   1:  PR[91,2] = PR[90,2] + -0.747;
   1:  PR[91,3] = PR[90,3] + 87.378;
   1:L PR[91] R[100]mm/sec CNT100;
   1:  PR[91,1] = PR[90,1] + -60.955;
   1:  PR[91,2] = PR[90,2] + -4.707;
   1:  PR[91,3] = PR[90,3] + 87.394;
   1:L PR[91] R[100]mm/sec CNT100;
   1:  PR[91,1] = PR[90,1] + -60.838;
   1:  PR[91,2] = PR[90,2] + -5.325;
   1:  PR[91,3] = PR[90,3] + 87.411;
   1:L PR[91] R[100]mm/sec CNT100;
   1:  PR[91,1] = PR[90,1] + -58.970;
   1:  PR[91,2] = PR[90,2] + -9.317;
   1:  PR[91,3] = PR[90,3] + 87.413;
   1:L PR[91] R[100]mm/sec CNT100;
   1:  PR[91,1] = PR[90,1] + -58.652;
   1:  PR[91,2] = PR[90,2] + -9.976;
   1:  PR[91,3] = PR[90,3] + 87.432;
   1:L PR[91] R[100]mm/sec CNT100;
   1:  PR[91,1] = PR[90,1] + -56.254;
   1:  PR[91,2] = PR[90,2] + -12.901;
   1:  PR[91,3] = PR[90,3] + 87.435;
   1:L PR[91] R[100]mm/sec CNT100;
   1:  PR[91,1] = PR[90,1] + -54.881;
   1:  PR[91,2] = PR[90,2] + -14.517;
   1:  PR[91,3] = PR[90,3] + 87.451;
   1:L PR[91] R[100]mm/sec CNT100;
   1:  PR[91,1] = PR[90,1] + -52.801;
   1:  PR[91,2] = PR[90,2] + -16.191;
   1:  PR[91,3] = PR[90,3] + 87.460;
   1:L PR[91] R[100]mm/sec CNT100;
   1:  PR[91,1] = PR[90,1] + -49.375;
   1:  PR[91,2] = PR[90,2] + -18.826;
   1:  PR[91,3] = PR[90,3] + 87.472;
   1:L PR[91] R[100]mm/sec CNT100;
   1:  PR[91,1] = PR[90,1] + -48.727;
   1:  PR[91,2] = PR[90,2] + -19.184;
   1:  PR[91,3] = PR[90,3] + 87.490;
   1:L PR[91] R[100]mm/sec CNT100;
   1:  PR[91,1] = PR[90,1] + -47.166;
   1:  PR[91,2] = PR[90,2] + -19.996;
   1:  PR[91,3] = PR[90,3] + 87.493;
   1:L PR[91] R[100]mm/sec CNT100;
   1:  PR[91,1] = PR[90,1] + -42.988;
   1:  PR[91,2] = PR[90,2] + -21.916;
   1:  PR[91,3] = PR[90,3] + 87.501;
   1:L PR[91] R[100]mm/sec CNT100;
   1:  PR[91,1] = PR[90,1] + -40.604;
   1:  PR[91,2] = PR[90,2] + -22.839;
   1:  PR[91,3] = PR[90,3] + 87.521;
   1:L PR[91] R[100]mm/sec CNT100;
   1:  PR[91,1] = PR[90,1] + -37.595;
   1:  PR[91,2] = PR[90,2] + -23.754;
   1:  PR[91,3] = PR[90,3] + 87.531;
   1:L PR[91] R[100]mm/sec CNT100;
   1:  PR[91,1] = PR[90,1] + -34.373;
   1:  PR[91,2] = PR[90,2] + -24.687;
   1:  PR[91,3] = PR[90,3] + 87.545;
   1:L PR[91] R[100]mm/sec CNT100;
   1:  PR[91,1] = PR[90,1] + -31.993;
   1:  PR[91,2] = PR[90,2] + -25.305;
   1:  PR[91,3] = PR[90,3] + 87.559;
   1:L PR[91] R[100]mm/sec CNT100;
   1:  PR[91,1] = PR[90,1] + -22.909;
   1:  PR[91,2] = PR[90,2] + -26.927;
   1:  PR[91,3] = PR[90,3] + 87.570;
   1:L PR[91] R[100]mm/sec CNT100;
   1:  PR[91,1] = PR[90,1] + -19.445;
   1:  PR[91,2] = PR[90,2] + -27.305;
   1:  PR[91,3] = PR[90,3] + 87.609;
   1:L PR[91] R[100]mm/sec CNT100;
   1:  PR[91,1] = PR[90,1] + -13.177;
   1:  PR[91,2] = PR[90,2] + -27.959;
   1:  PR[91,3] = PR[90,3] + 87.624;
   1:L PR[91] R[100]mm/sec CNT100;
   1:  PR[91,1] = PR[90,1] + -6.530;
   1:  PR[91,2] = PR[90,2] + -28.215;
   1:  PR[91,3] = PR[90,3] + 87.651;
   1:L PR[91] R[100]mm/sec CNT100;
   1:  PR[91,1] = PR[90,1] + -2.969;
   1:  PR[91,2] = PR[90,2] + -28.333;
   1:  PR[91,3] = PR[90,3] + 87.679;
   1:L PR[91] R[100]mm/sec CNT100;
   1:  PR[91,1] = PR[90,1] + 7.766;
   1:  PR[91,2] = PR[90,2] + -27.986;
   1:  PR[91,3] = PR[90,3] + 87.694;
   1:L PR[91] R[100]mm/sec CNT100;
   1:  PR[91,1] = PR[90,1] + 9.166;
   1:  PR[91,2] = PR[90,2] + -28.006;
   1:  PR[91,3] = PR[90,3] + 87.740;
   1:L PR[91] R[100]mm/sec CNT100;
   1:  PR[91,1] = PR[90,1] + 10.864;
   1:  PR[91,2] = PR[90,2] + -27.971;
   1:  PR[91,3] = PR[90,3] + 87.746;
   1:L PR[91] R[100]mm/sec CNT100;
   1:  PR[91,1] = PR[90,1] + 12.500;
   1:  PR[91,2] = PR[90,2] + -27.879;
   1:  PR[91,3] = PR[90,3] + 87.753;
   1:L PR[91] R[100]mm/sec CNT100;
   1:  PR[91,1] = PR[90,1] + 13.907;
   1:  PR[91,2] = PR[90,2] + -27.767;
   1:  PR[91,3] = PR[90,3] + 87.760;
   1:L PR[91] R[100]mm/sec CNT100;
   1:  PR[91,1] = PR[90,1] + 17.964;
   1:  PR[91,2] = PR[90,2] + -28.256;
   1:  PR[91,3] = PR[90,3] + 87.766;
   1:L PR[91] R[100]mm/sec CNT100;
   1:  PR[91,1] = PR[90,1] + 18.028;
   1:  PR[91,2] = PR[90,2] + -28.259;
   1:  PR[91,3] = PR[90,3] + 87.784;
   1:L PR[91] R[100]mm/sec CNT100;
   1:  PR[91,1] = PR[90,1] + 23.535;
   1:  PR[91,2] = PR[90,2] + -28.156;
   1:L PR[91] R[100]mm/sec CNT100;
   1:  PR[91,1] = PR[90,1] + 23.597;
   1:  PR[91,2] = PR[90,2] + -28.531;
   1:  PR[91,3] = PR[90,3] + 87.808;
   1:L PR[91] R[100]mm/sec CNT100;
   1:  PR[91,1] = PR[90,1] + 23.842;
   1:  PR[91,2] = PR[90,2] + -28.584;
   1:  PR[91,3] = PR[90,3] + 87.809;
   1:L PR[91] R[100]mm/sec CNT100;
   1:  PR[91,1] = PR[90,1] + 27.676;
   1:  PR[91,2] = PR[90,2] + -29.474;
   1:  PR[91,3] = PR[90,3] + 87.810;
   1:L PR[91] R[100]mm/sec CNT100;
   1:  PR[91,1] = PR[90,1] + 32.886;
   1:  PR[91,2] = PR[90,2] + -29.769;
   1:  PR[91,3] = PR[90,3] + 87.827;
   1:L PR[91] R[100]mm/sec CNT100;
   1:  PR[91,1] = PR[90,1] + 38.004;
   1:  PR[91,2] = PR[90,2] + -29.151;
   1:  PR[91,3] = PR[90,3] + 87.849;
   1:L PR[91] R[100]mm/sec CNT100;
   1:  PR[91,1] = PR[90,1] + 42.904;
   1:  PR[91,2] = PR[90,2] + -27.658;
   1:  PR[91,3] = PR[90,3] + 87.871;
   1:L PR[91] R[100]mm/sec CNT100;
   1:  PR[91,1] = PR[90,1] + 47.549;
   1:  PR[91,2] = PR[90,2] + -25.414;
   1:  PR[91,3] = PR[90,3] + 87.893;
   1:L PR[91] R[100]mm/sec CNT100;
   1:  PR[91,1] = PR[90,1] + 51.641;
   1:  PR[91,2] = PR[90,2] + -22.484;
   1:  PR[91,3] = PR[90,3] + 87.915;
   1:L PR[91] R[100]mm/sec CNT100;
   1:  PR[91,1] = PR[90,1] + 54.090;
   1:  PR[91,2] = PR[90,2] + -19.978;
   1:  PR[91,3] = PR[90,3] + 87.937;
   1:L PR[91] R[100]mm/sec CNT100;
   1:  PR[91,1] = PR[90,1] + 55.118;
   1:  PR[91,2] = PR[90,2] + -19.051;
   1:  PR[91,3] = PR[90,3] + 87.952;
   1:L PR[91] R[100]mm/sec CNT100;
   1:  PR[91,1] = PR[90,1] + 55.443;
   1:  PR[91,2] = PR[90,2] + -18.712;
   1:  PR[91,3] = PR[90,3] + 87.957;
   1:L PR[91] R[100]mm/sec CNT100;
   1:  PR[91,1] = PR[90,1] + 57.489;
   1:  PR[91,2] = PR[90,2] + -16.058;
   1:  PR[91,3] = PR[90,3] + 87.960;
   1:L PR[91] R[100]mm/sec CNT100;
   1:  PR[91,1] = PR[90,1] + 58.739;
   1:  PR[91,2] = PR[90,2] + -14.217;
   1:  PR[91,3] = PR[90,3] + 87.974;
   1:L PR[91] R[100]mm/sec CNT100;
   1:  PR[91,1] = PR[90,1] + 59.321;
   1:  PR[91,2] = PR[90,2] + -13.077;
   1:  PR[91,3] = PR[90,3] + 87.983;
   1:L PR[91] R[100]mm/sec CNT100;
   1:  PR[91,1] = PR[90,1] + 60.647;
   1:  PR[91,2] = PR[90,2] + -10.162;
   1:  PR[91,3] = PR[90,3] + 87.989;
   1:L PR[91] R[100]mm/sec CNT100;
   1:  PR[91,1] = PR[90,1] + 60.947;
   1:  PR[91,2] = PR[90,2] + -9.626;
   1:  PR[91,3] = PR[90,3] + 88.002;
   1:L PR[91] R[100]mm/sec CNT100;
   1:  PR[91,1] = PR[90,1] + 60.967;
   1:  PR[91,2] = PR[90,2] + -9.586;
   1:  PR[91,3] = PR[90,3] + 88.005;
   1:L PR[91] R[100]mm/sec CNT100;
   1:  PR[91,1] = PR[90,1] + 62.074;
   1:  PR[91,2] = PR[90,2] + -6.140;
   1:L PR[91] R[100]mm/sec CNT100;
   1:  PR[91,1] = PR[90,1] + 62.374;
   1:  PR[91,2] = PR[90,2] + -5.080;
   1:  PR[91,3] = PR[90,3] + 88.021;
   1:L PR[91] R[100]mm/sec CNT100;
   1:  PR[91,1] = PR[90,1] + 62.812;
   1:  PR[91,2] = PR[90,2] + -0.723;
   1:  PR[91,3] = PR[90,3] + 88.025;
   1:L PR[91] R[100]mm/sec CNT100;
   1:  PR[91,1] = PR[90,1] + 62.655;
   1:  PR[91,2] = PR[90,2] + 0.936;
   1:  PR[91,3] = PR[90,3] + 88.044;
   1:L PR[91] R[100]mm/sec CNT100;
   1:  PR[91,1] = PR[90,1] + 62.375;
   1:  PR[91,2] = PR[90,2] + 3.618;
   1:  PR[91,3] = PR[90,3] + 88.051;
   1:L PR[91] R[100]mm/sec CNT100;
   1:  PR[91,1] = PR[90,1] + 62.074;
   1:  PR[91,2] = PR[90,2] + 4.681;
   1:  PR[91,3] = PR[90,3] + 88.063;
   1:L PR[91] R[100]mm/sec CNT100;
   1:  PR[91,1] = PR[90,1] + 60.967;
   1:  PR[91,2] = PR[90,2] + 8.127;
   1:  PR[91,3] = PR[90,3] + 88.067;
   1:L PR[91] R[100]mm/sec CNT100;
   1:  PR[91,1] = PR[90,1] + 60.947;
   1:  PR[91,2] = PR[90,2] + 8.167;
   1:  PR[91,3] = PR[90,3] + 88.083;
   1:L PR[91] R[100]mm/sec CNT100;
   1:  PR[91,1] = PR[90,1] + 60.647;
   1:  PR[91,2] = PR[90,2] + 8.703;
   1:L PR[91] R[100]mm/sec CNT100;
   1:  PR[91,1] = PR[90,1] + 59.321;
   1:  PR[91,2] = PR[90,2] + 11.618;
   1:  PR[91,3] = PR[90,3] + 88.086;
   1:L PR[91] R[100]mm/sec CNT100;
   1:  PR[91,1] = PR[90,1] + 58.739;
   1:  PR[91,2] = PR[90,2] + 12.758;
   1:  PR[91,3] = PR[90,3] + 88.099;
   1:L PR[91] R[100]mm/sec CNT100;
   1:  PR[91,1] = PR[90,1] + 57.489;
   1:  PR[91,2] = PR[90,2] + 14.600;
   1:  PR[91,3] = PR[90,3] + 88.105;
   1:L PR[91] R[100]mm/sec CNT100;
   1:  PR[91,1] = PR[90,1] + 55.443;
   1:  PR[91,2] = PR[90,2] + 17.253;
   1:  PR[91,3] = PR[90,3] + 88.114;
   1:L PR[91] R[100]mm/sec CNT100;
   1:  PR[91,1] = PR[90,1] + 55.118;
   1:  PR[91,2] = PR[90,2] + 17.592;
   1:  PR[91,3] = PR[90,3] + 88.129;
   1:L PR[91] R[100]mm/sec CNT100;
   1:  PR[91,1] = PR[90,1] + 54.090;
   1:  PR[91,2] = PR[90,2] + 18.519;
   1:  PR[91,3] = PR[90,3] + 88.131;
   1:L PR[91] R[100]mm/sec CNT100;
   1:  PR[91,1] = PR[90,1] + 51.641;
   1:  PR[91,2] = PR[90,2] + 21.026;
   1:  PR[91,3] = PR[90,3] + 88.136;
   1:L PR[91] R[100]mm/sec CNT100;
   1:  PR[91,1] = PR[90,1] + 47.549;
   1:  PR[91,2] = PR[90,2] + 23.955;
   1:  PR[91,3] = PR[90,3] + 88.151;
   1:L PR[91] R[100]mm/sec CNT100;
   1:  PR[91,1] = PR[90,1] + 42.904;
   1:  PR[91,2] = PR[90,2] + 26.199;
   1:  PR[91,3] = PR[90,3] + 88.173;
   1:L PR[91] R[100]mm/sec CNT100;
   1:  PR[91,1] = PR[90,1] + 38.004;
   1:  PR[91,2] = PR[90,2] + 27.692;
   1:  PR[91,3] = PR[90,3] + 88.195;
   1:L PR[91] R[100]mm/sec CNT100;
   1:  PR[91,1] = PR[90,1] + 32.886;
   1:  PR[91,2] = PR[90,2] + 28.310;
   1:  PR[91,3] = PR[90,3] + 88.217;
   1:L PR[91] R[100]mm/sec CNT100;
   1:  PR[91,1] = PR[90,1] + 27.676;
   1:  PR[91,2] = PR[90,2] + 28.015;
   1:  PR[91,3] = PR[90,3] + 88.239;
   1:L PR[91] R[100]mm/sec CNT100;
   1:  PR[91,1] = PR[90,1] + 23.842;
   1:  PR[91,2] = PR[90,2] + 27.125;
   1:  PR[91,3] = PR[90,3] + 88.261;
   1:L PR[91] R[100]mm/sec CNT100;
   1:  PR[91,1] = PR[90,1] + 22.019;
   1:  PR[91,2] = PR[90,2] + 26.732;
   1:  PR[91,3] = PR[90,3] + 88.278;
   1:L PR[91] R[100]mm/sec CNT100;
   1:  PR[91,1] = PR[90,1] + 18.496;
   1:  PR[91,2] = PR[90,2] + 26.796;
   1:  PR[91,3] = PR[90,3] + 88.286;
   1:L PR[91] R[100]mm/sec CNT100;
   1:  PR[91,1] = PR[90,1] + 17.924;
   1:  PR[91,2] = PR[90,2] + 26.793;
   1:  PR[91,3] = PR[90,3] + 88.301;
   1:L PR[91] R[100]mm/sec CNT100;
   1:  PR[91,1] = PR[90,1] + 13.907;
   1:  PR[91,2] = PR[90,2] + 26.308;
   1:  PR[91,3] = PR[90,3] + 88.303;
   1:L PR[91] R[100]mm/sec CNT100;
   1:  PR[91,1] = PR[90,1] + 12.500;
   1:  PR[91,2] = PR[90,2] + 26.420;
   1:  PR[91,3] = PR[90,3] + 88.320;
   1:L PR[91] R[100]mm/sec CNT100;
   1:  PR[91,1] = PR[90,1] + 10.887;
   1:  PR[91,2] = PR[90,2] + 26.511;
   1:  PR[91,3] = PR[90,3] + 88.326;
   1:L PR[91] R[100]mm/sec CNT100;
   1:  PR[91,1] = PR[90,1] + 8.242;
   1:  PR[91,2] = PR[90,2] + 26.490;
   1:  PR[91,3] = PR[90,3] + 88.333;
   1:L PR[91] R[100]mm/sec CNT100;
   1:  PR[91,1] = PR[90,1] + 6.900;
   1:  PR[91,2] = PR[90,2] + 26.563;
   1:  PR[91,3] = PR[90,3] + 88.345;
   1:L PR[91] R[100]mm/sec CNT100;
   1:  PR[91,1] = PR[90,1] + -2.968;
   1:  PR[91,2] = PR[90,2] + 26.874;
   1:  PR[91,3] = PR[90,3] + 88.350;
   1:L PR[91] R[100]mm/sec CNT100;
   1:  PR[91,1] = PR[90,1] + -6.530;
   1:  PR[91,2] = PR[90,2] + 26.756;
   1:  PR[91,3] = PR[90,3] + 88.392;
   1:L PR[91] R[100]mm/sec CNT100;
   1:  PR[91,1] = PR[90,1] + -13.177;
   1:  PR[91,2] = PR[90,2] + 26.500;
   1:  PR[91,3] = PR[90,3] + 88.408;
   1:L PR[91] R[100]mm/sec CNT100;
   1:  PR[91,1] = PR[90,1] + -19.445;
   1:  PR[91,2] = PR[90,2] + 25.846;
   1:  PR[91,3] = PR[90,3] + 88.436;
   1:L PR[91] R[100]mm/sec CNT100;
   1:  PR[91,1] = PR[90,1] + -22.909;
   1:  PR[91,2] = PR[90,2] + 25.468;
   1:  PR[91,3] = PR[90,3] + 88.463;
   1:L PR[91] R[100]mm/sec CNT100;
   1:  PR[91,1] = PR[90,1] + -31.993;
   1:  PR[91,2] = PR[90,2] + 23.847;
   1:  PR[91,3] = PR[90,3] + 88.478;
   1:L PR[91] R[100]mm/sec CNT100;
   1:  PR[91,1] = PR[90,1] + -34.366;
   1:  PR[91,2] = PR[90,2] + 23.230;
   1:  PR[91,3] = PR[90,3] + 88.517;
   1:L PR[91] R[100]mm/sec CNT100;
   1:  PR[91,1] = PR[90,1] + -41.010;
   1:  PR[91,2] = PR[90,2] + 21.258;
   1:  PR[91,3] = PR[90,3] + 88.528;
   1:L PR[91] R[100]mm/sec CNT100;
   1:  PR[91,1] = PR[90,1] + -42.927;
   1:  PR[91,2] = PR[90,2] + 20.525;
   1:  PR[91,3] = PR[90,3] + 88.557;
   1:L PR[91] R[100]mm/sec CNT100;
   1:  PR[91,1] = PR[90,1] + -45.770;
   1:  PR[91,2] = PR[90,2] + 19.214;
   1:  PR[91,3] = PR[90,3] + 88.566;
   1:L PR[91] R[100]mm/sec CNT100;
   1:  PR[91,1] = PR[90,1] + -49.044;
   1:  PR[91,2] = PR[90,2] + 17.545;
   1:  PR[91,3] = PR[90,3] + 88.579;
   1:L PR[91] R[100]mm/sec CNT100;
   1:  PR[91] = PR[90];
   1:  PR[91,1] = PR[90,1] + -52.926;
   1:  PR[91,2] = PR[90,2] + 13.640;
   1:  PR[91,3] = PR[90,3] + 89.895;
   1:L PR[91] R[100]mm/sec CNT100;
   1:  PR[91,1] = PR[90,1] + -56.042;
   1:  PR[91,2] = PR[90,2] + 10.206;
   1:  PR[91,3] = PR[90,3] + 88.619;
   1:L PR[91] R[100]mm/sec CNT100;
   1:  PR[91,1] = PR[90,1] + -56.949;
   1:  PR[91,2] = PR[90,2] + 9.159;
   1:  PR[91,3] = PR[90,3] + 88.639;
   1:L PR[91] R[100]mm/sec CNT100;
   1:  PR[91,1] = PR[90,1] + -59.443;
   1:  PR[91,2] = PR[90,2] + 4.317;
   1:  PR[91,3] = PR[90,3] + 88.645;
   1:L PR[91] R[100]mm/sec CNT100;
   1:  PR[91,1] = PR[90,1] + -59.446;
   1:  PR[91,2] = PR[90,2] + 4.299;
   1:  PR[91,3] = PR[90,3] + 88.668;
   1:L PR[91] R[100]mm/sec CNT100;
   1:  PR[91,1] = PR[90,1] + -60.232;
   1:  PR[91,2] = PR[90,2] + -0.740;
   1:L PR[91] R[100]mm/sec CNT100;
   1:  PR[91,1] = PR[90,1] + -60.086;
   1:  PR[91,2] = PR[90,2] + -1.741;
   1:  PR[91,3] = PR[90,3] + 88.690;
   1:L PR[91] R[100]mm/sec CNT100;
   1:  PR[91,1] = PR[90,1] + -59.602;
   1:  PR[91,2] = PR[90,2] + -4.260;
   1:  PR[91,3] = PR[90,3] + 88.695;
   1:L PR[91] R[100]mm/sec CNT100;
   1:  PR[91,1] = PR[90,1] + -59.526;
   1:  PR[91,2] = PR[90,2] + -4.467;
   1:  PR[91,3] = PR[90,3] + 88.706;
   1:L PR[91] R[100]mm/sec CNT100;
   1:  PR[91,1] = PR[90,1] + -59.377;
   1:  PR[91,2] = PR[90,2] + -5.416;
   1:  PR[91,3] = PR[90,3] + 88.707;
   1:L PR[91] R[100]mm/sec CNT100;
   1:  PR[91,1] = PR[90,1] + -57.834;
   1:  PR[91,2] = PR[90,2] + -8.715;
   1:  PR[91,3] = PR[90,3] + 88.711;
   1:L PR[91] R[100]mm/sec CNT100;
   1:  PR[91,1] = PR[90,1] + -57.168;
   1:  PR[91,2] = PR[90,2] + -10.096;
   1:  PR[91,3] = PR[90,3] + 88.727;
   1:L PR[91] R[100]mm/sec CNT100;
   1:  PR[91,1] = PR[90,1] + -55.257;
   1:  PR[91,2] = PR[90,2] + -12.427;
   1:  PR[91,3] = PR[90,3] + 88.733;
   1:L PR[91] R[100]mm/sec CNT100;
   1:  PR[91,1] = PR[90,1] + -53.331;
   1:  PR[91,2] = PR[90,2] + -14.694;
   1:  PR[91,3] = PR[90,3] + 88.746;
   1:L PR[91] R[100]mm/sec CNT100;
   1:  PR[91,1] = PR[90,1] + -51.908;
   1:  PR[91,2] = PR[90,2] + -15.839;
   1:  PR[91,3] = PR[90,3] + 88.759;
   1:L PR[91] R[100]mm/sec CNT100;
   1:  PR[91,1] = PR[90,1] + -47.806;
   1:  PR[91,2] = PR[90,2] + -18.993;
   1:  PR[91,3] = PR[90,3] + 88.767;
   1:L PR[91] R[100]mm/sec CNT100;
   1:  PR[91,1] = PR[90,1] + -41.701;
   1:  PR[91,2] = PR[90,2] + -21.799;
   1:  PR[91,3] = PR[90,3] + 88.789;
   1:L PR[91] R[100]mm/sec CNT100;
   1:  PR[91,1] = PR[90,1] + -38.057;
   1:  PR[91,2] = PR[90,2] + -23.210;
   1:  PR[91,3] = PR[90,3] + 88.818;
   1:L PR[91] R[100]mm/sec CNT100;
   1:  PR[91,1] = PR[90,1] + -36.603;
   1:  PR[91,2] = PR[90,2] + -23.652;
   1:  PR[91,3] = PR[90,3] + 88.835;
   1:L PR[91] R[100]mm/sec CNT100;
   1:  PR[91,1] = PR[90,1] + -35.021;
   1:  PR[91,2] = PR[90,2] + -24.110;
   1:  PR[91,3] = PR[90,3] + 88.842;
   1:L PR[91] R[100]mm/sec CNT100;
   1:  PR[91,1] = PR[90,1] + -29.592;
   1:  PR[91,2] = PR[90,2] + -25.521;
   1:  PR[91,3] = PR[90,3] + 88.849;
   1:L PR[91] R[100]mm/sec CNT100;
   1:  PR[91,1] = PR[90,1] + -20.438;
   1:  PR[91,2] = PR[90,2] + -27.159;
   1:  PR[91,3] = PR[90,3] + 88.873;
   1:L PR[91] R[100]mm/sec CNT100;
   1:  PR[91,1] = PR[90,1] + -16.033;
   1:  PR[91,2] = PR[90,2] + -27.640;
   1:  PR[91,3] = PR[90,3] + 88.913;
   1:L PR[91] R[100]mm/sec CNT100;
   1:  PR[91,1] = PR[90,1] + -10.631;
   1:  PR[91,2] = PR[90,2] + -28.203;
   1:  PR[91,3] = PR[90,3] + 88.932;
   1:L PR[91] R[100]mm/sec CNT100;
   1:  PR[91,1] = PR[90,1] + -2.987;
   1:  PR[91,2] = PR[90,2] + -28.498;
   1:  PR[91,3] = PR[90,3] + 88.956;
   1:L PR[91] R[100]mm/sec CNT100;
   1:  PR[91,1] = PR[90,1] + -0.342;
   1:  PR[91,2] = PR[90,2] + -28.586;
   1:  PR[91,3] = PR[90,3] + 88.989;
   1:L PR[91] R[100]mm/sec CNT100;
   1:  PR[91,1] = PR[90,1] + 9.329;
   1:  PR[91,2] = PR[90,2] + -28.281;
   1:  PR[91,3] = PR[90,3] + 89.000;
   1:L PR[91] R[100]mm/sec CNT100;
   1:  PR[91,1] = PR[90,1] + 10.609;
   1:  PR[91,2] = PR[90,2] + -28.228;
   1:  PR[91,3] = PR[90,3] + 89.042;
   1:L PR[91] R[100]mm/sec CNT100;
   1:  PR[91,1] = PR[90,1] + 11.898;
   1:  PR[91,2] = PR[90,2] + -28.202;
   1:  PR[91,3] = PR[90,3] + 89.047;
   1:L PR[91] R[100]mm/sec CNT100;
   1:  PR[91,1] = PR[90,1] + 13.967;
   1:  PR[91,2] = PR[90,2] + -28.086;
   1:  PR[91,3] = PR[90,3] + 89.053;
   1:L PR[91] R[100]mm/sec CNT100;
   1:  PR[91,1] = PR[90,1] + 14.757;
   1:  PR[91,2] = PR[90,2] + -28.023;
   1:  PR[91,3] = PR[90,3] + 89.062;
   1:L PR[91] R[100]mm/sec CNT100;
   1:  PR[91,1] = PR[90,1] + 16.691;
   1:  PR[91,2] = PR[90,2] + -28.260;
   1:  PR[91,3] = PR[90,3] + 89.065;
   1:L PR[91] R[100]mm/sec CNT100;
   1:  PR[91,1] = PR[90,1] + 18.052;
   1:  PR[91,2] = PR[90,2] + -28.399;
   1:  PR[91,3] = PR[90,3] + 89.074;
   1:L PR[91] R[100]mm/sec CNT100;
   1:  PR[91,1] = PR[90,1] + 18.662;
   1:  PR[91,2] = PR[90,2] + -28.427;
   1:  PR[91,3] = PR[90,3] + 89.079;
   1:L PR[91] R[100]mm/sec CNT100;
   1:  PR[91,1] = PR[90,1] + 23.335;
   1:  PR[91,2] = PR[90,2] + -28.340;
   1:  PR[91,3] = PR[90,3] + 89.082;
   1:L PR[91] R[100]mm/sec CNT100;
   1:  PR[91,1] = PR[90,1] + 23.411;
   1:  PR[91,2] = PR[90,2] + -28.745;
   1:  PR[91,3] = PR[90,3] + 89.102;
   1:L PR[91] R[100]mm/sec CNT100;
   1:  PR[91,1] = PR[90,1] + 27.421;
   1:  PR[91,2] = PR[90,2] + -29.668;
   1:  PR[91,3] = PR[90,3] + 89.104;
   1:L PR[91] R[100]mm/sec CNT100;
   1:  PR[91,1] = PR[90,1] + 32.665;
   1:  PR[91,2] = PR[90,2] + -29.960;
   1:  PR[91,3] = PR[90,3] + 89.122;
   1:L PR[91] R[100]mm/sec CNT100;
   1:  PR[91,1] = PR[90,1] + 37.819;
   1:  PR[91,2] = PR[90,2] + -29.339;
   1:  PR[91,3] = PR[90,3] + 89.144;
   1:L PR[91] R[100]mm/sec CNT100;
   1:  PR[91,1] = PR[90,1] + 42.716;
   1:  PR[91,2] = PR[90,2] + -27.843;
   1:  PR[91,3] = PR[90,3] + 89.167;
   1:L PR[91] R[100]mm/sec CNT100;
   1:  PR[91,1] = PR[90,1] + 45.674;
   1:  PR[91,2] = PR[90,2] + -26.321;
   1:  PR[91,3] = PR[90,3] + 89.189;
   1:L PR[91] R[100]mm/sec CNT100;
   1:  PR[91,1] = PR[90,1] + 47.308;
   1:  PR[91,2] = PR[90,2] + -25.531;
   1:  PR[91,3] = PR[90,3] + 89.203;
   1:L PR[91] R[100]mm/sec CNT100;
   1:  PR[91,1] = PR[90,1] + 51.432;
   1:  PR[91,2] = PR[90,2] + -22.575;
   1:  PR[91,3] = PR[90,3] + 89.211;
   1:L PR[91] R[100]mm/sec CNT100;
   1:  PR[91,1] = PR[90,1] + 54.911;
   1:  PR[91,2] = PR[90,2] + -19.016;
   1:  PR[91,3] = PR[90,3] + 89.233;
   1:L PR[91] R[100]mm/sec CNT100;
   1:  PR[91,1] = PR[90,1] + 56.172;
   1:  PR[91,2] = PR[90,2] + -17.160;
   1:  PR[91,3] = PR[90,3] + 89.254;
   1:L PR[91] R[100]mm/sec CNT100;
   1:  PR[91,1] = PR[90,1] + 57.617;
   1:  PR[91,2] = PR[90,2] + -15.286;
   1:  PR[91,3] = PR[90,3] + 89.264;
   1:L PR[91] R[100]mm/sec CNT100;
   1:  PR[91,1] = PR[90,1] + 58.051;
   1:  PR[91,2] = PR[90,2] + -14.646;
   1:  PR[91,3] = PR[90,3] + 89.274;
   1:L PR[91] R[100]mm/sec CNT100;
   1:  PR[91,1] = PR[90,1] + 59.413;
   1:  PR[91,2] = PR[90,2] + -11.978;
   1:  PR[91,3] = PR[90,3] + 89.278;
   1:L PR[91] R[100]mm/sec CNT100;
   1:  PR[91,1] = PR[90,1] + 60.325;
   1:  PR[91,2] = PR[90,2] + -9.973;
   1:  PR[91,3] = PR[90,3] + 89.291;
   1:L PR[91] R[100]mm/sec CNT100;
   1:  PR[91,1] = PR[90,1] + 60.726;
   1:  PR[91,2] = PR[90,2] + -8.594;
   1:  PR[91,3] = PR[90,3] + 89.300;
   1:L PR[91] R[100]mm/sec CNT100;
   1:  PR[91,1] = PR[90,1] + 61.580;
   1:  PR[91,2] = PR[90,2] + -5.335;
   1:  PR[91,3] = PR[90,3] + 89.306;
   1:L PR[91] R[100]mm/sec CNT100;
   1:  PR[91,1] = PR[90,1] + 61.980;
   1:  PR[91,2] = PR[90,2] + -0.770;
   1:  PR[91,3] = PR[90,3] + 89.321;
   1:L PR[91] R[100]mm/sec CNT100;
   1:  PR[91,1] = PR[90,1] + 61.703;
   1:  PR[91,2] = PR[90,2] + 2.215;
   1:  PR[91,3] = PR[90,3] + 89.341;
   1:L PR[91] R[100]mm/sec CNT100;
   1:  PR[91,1] = PR[90,1] + 61.577;
   1:  PR[91,2] = PR[90,2] + 3.888;
   1:  PR[91,3] = PR[90,3] + 89.354;
   1:L PR[91] R[100]mm/sec CNT100;
   1:  PR[91,1] = PR[90,1] + 60.726;
   1:  PR[91,2] = PR[90,2] + 7.135;
   1:  PR[91,3] = PR[90,3] + 89.361;
   1:L PR[91] R[100]mm/sec CNT100;
   1:  PR[91,1] = PR[90,1] + 60.325;
   1:  PR[91,2] = PR[90,2] + 8.514;
   1:  PR[91,3] = PR[90,3] + 89.375;
   1:L PR[91] R[100]mm/sec CNT100;
   1:  PR[91,1] = PR[90,1] + 59.413;
   1:  PR[91,2] = PR[90,2] + 10.519;
   1:  PR[91,3] = PR[90,3] + 89.381;
   1:L PR[91] R[100]mm/sec CNT100;
   1:  PR[91,1] = PR[90,1] + 58.051;
   1:  PR[91,2] = PR[90,2] + 13.187;
   1:  PR[91,3] = PR[90,3] + 89.391;
   1:L PR[91] R[100]mm/sec CNT100;
   1:  PR[91,1] = PR[90,1] + 57.617;
   1:  PR[91,2] = PR[90,2] + 13.827;
   1:  PR[91,3] = PR[90,3] + 89.404;
   1:L PR[91] R[100]mm/sec CNT100;
   1:  PR[91,1] = PR[90,1] + 56.172;
   1:  PR[91,2] = PR[90,2] + 15.701;
   1:  PR[91,3] = PR[90,3] + 89.407;
   1:L PR[91] R[100]mm/sec CNT100;
   1:  PR[91,1] = PR[90,1] + 54.911;
   1:  PR[91,2] = PR[90,2] + 17.557;
   1:  PR[91,3] = PR[90,3] + 89.417;
   1:L PR[91] R[100]mm/sec CNT100;
   1:  PR[91,1] = PR[90,1] + 51.432;
   1:  PR[91,2] = PR[90,2] + 21.116;
   1:  PR[91,3] = PR[90,3] + 89.427;
   1:L PR[91] R[100]mm/sec CNT100;
   1:  PR[91,1] = PR[90,1] + 47.308;
   1:  PR[91,2] = PR[90,2] + 24.072;
   1:  PR[91,3] = PR[90,3] + 89.449;
   1:L PR[91] R[100]mm/sec CNT100;
   1:  PR[91,1] = PR[90,1] + 45.674;
   1:  PR[91,2] = PR[90,2] + 24.862;
   1:  PR[91,3] = PR[90,3] + 89.470;
   1:L PR[91] R[100]mm/sec CNT100;
   1:  PR[91,1] = PR[90,1] + 42.716;
   1:  PR[91,2] = PR[90,2] + 26.384;
   1:  PR[91,3] = PR[90,3] + 89.478;
   1:L PR[91] R[100]mm/sec CNT100;
   1:  PR[91,1] = PR[90,1] + 37.819;
   1:  PR[91,2] = PR[90,2] + 27.880;
   1:  PR[91,3] = PR[90,3] + 89.493;
   1:L PR[91] R[100]mm/sec CNT100;
   1:  PR[91,1] = PR[90,1] + 32.665;
   1:  PR[91,2] = PR[90,2] + 28.501;
   1:  PR[91,3] = PR[90,3] + 89.515;
   1:L PR[91] R[100]mm/sec CNT100;
   1:  PR[91,1] = PR[90,1] + 27.421;
   1:  PR[91,2] = PR[90,2] + 28.210;
   1:  PR[91,3] = PR[90,3] + 89.537;
   1:L PR[91] R[100]mm/sec CNT100;
   1:  PR[91,1] = PR[90,1] + 21.849;
   1:  PR[91,2] = PR[90,2] + 26.926;
   1:  PR[91,3] = PR[90,3] + 89.560;
   1:L PR[91] R[100]mm/sec CNT100;
   1:  PR[91,1] = PR[90,1] + 18.668;
   1:  PR[91,2] = PR[90,2] + 26.969;
   1:  PR[91,3] = PR[90,3] + 89.584;
   1:L PR[91] R[100]mm/sec CNT100;
   1:  PR[91,1] = PR[90,1] + 18.073;
   1:  PR[91,2] = PR[90,2] + 26.941;
   1:  PR[91,3] = PR[90,3] + 89.598;
   1:L PR[91] R[100]mm/sec CNT100;
   1:  PR[91,1] = PR[90,1] + 15.356;
   1:  PR[91,2] = PR[90,2] + 26.609;
   1:  PR[91,3] = PR[90,3] + 89.601;
   1:L PR[91] R[100]mm/sec CNT100;
   1:  PR[91,1] = PR[90,1] + 14.693;
   1:  PR[91,2] = PR[90,2] + 26.569;
   1:  PR[91,3] = PR[90,3] + 89.612;
   1:L PR[91] R[100]mm/sec CNT100;
   1:  PR[91,1] = PR[90,1] + 13.967;
   1:  PR[91,2] = PR[90,2] + 26.627;
   1:  PR[91,3] = PR[90,3] + 89.615;
   1:L PR[91] R[100]mm/sec CNT100;
   1:  PR[91,1] = PR[90,1] + 11.919;
   1:  PR[91,2] = PR[90,2] + 26.742;
   1:  PR[91,3] = PR[90,3] + 89.619;
   1:L PR[91] R[100]mm/sec CNT100;
   1:  PR[91,1] = PR[90,1] + 11.052;
   1:  PR[91,2] = PR[90,2] + 26.735;
   1:  PR[91,3] = PR[90,3] + 89.627;
   1:L PR[91] R[100]mm/sec CNT100;
   1:  PR[91,1] = PR[90,1] + 10.556;
   1:  PR[91,2] = PR[90,2] + 26.772;
   1:  PR[91,3] = PR[90,3] + 89.631;
   1:L PR[91] R[100]mm/sec CNT100;
   1:  PR[91,1] = PR[90,1] + 9.329;
   1:  PR[91,2] = PR[90,2] + 26.822;
   1:  PR[91,3] = PR[90,3] + 89.633;
   1:L PR[91] R[100]mm/sec CNT100;
   1:  PR[91,1] = PR[90,1] + -0.341;
   1:  PR[91,2] = PR[90,2] + 27.127;
   1:  PR[91,3] = PR[90,3] + 89.639;
   1:L PR[91] R[100]mm/sec CNT100;
   1:  PR[91,1] = PR[90,1] + -2.989;
   1:  PR[91,2] = PR[90,2] + 27.039;
   1:  PR[91,3] = PR[90,3] + 89.680;
   1:L PR[91] R[100]mm/sec CNT100;
   1:  PR[91,1] = PR[90,1] + -10.631;
   1:  PR[91,2] = PR[90,2] + 26.744;
   1:  PR[91,3] = PR[90,3] + 89.692;
   1:L PR[91] R[100]mm/sec CNT100;
   1:  PR[91,1] = PR[90,1] + -16.033;
   1:  PR[91,2] = PR[90,2] + 26.181;
   1:  PR[91,3] = PR[90,3] + 89.725;
   1:L PR[91] R[100]mm/sec CNT100;
   1:  PR[91,1] = PR[90,1] + -20.438;
   1:  PR[91,2] = PR[90,2] + 25.700;
   1:  PR[91,3] = PR[90,3] + 89.748;
   1:L PR[91] R[100]mm/sec CNT100;
   1:  PR[91,1] = PR[90,1] + -29.592;
   1:  PR[91,2] = PR[90,2] + 24.062;
   1:  PR[91,3] = PR[90,3] + 89.767;
   1:L PR[91] R[100]mm/sec CNT100;
   1:  PR[91,1] = PR[90,1] + -35.015;
   1:  PR[91,2] = PR[90,2] + 22.653;
   1:  PR[91,3] = PR[90,3] + 89.807;
   1:L PR[91] R[100]mm/sec CNT100;
   1:  PR[91,1] = PR[90,1] + -38.264;
   1:  PR[91,2] = PR[90,2] + 21.688;
   1:  PR[91,3] = PR[90,3] + 89.832;
   1:L PR[91] R[100]mm/sec CNT100;
   1:  PR[91,1] = PR[90,1] + -41.654;
   1:  PR[91,2] = PR[90,2] + 20.393;
   1:  PR[91,3] = PR[90,3] + 89.846;
   1:L PR[91] R[100]mm/sec CNT100;
   1:  PR[91,1] = PR[90,1] + -46.607;
   1:  PR[91,2] = PR[90,2] + 18.108;
   1:  PR[91,3] = PR[90,3] + 89.862;
   1:L PR[91] R[100]mm/sec CNT100;
   1:  PR[91,1] = PR[90,1] + -47.701;
   1:  PR[91,2] = PR[90,2] + 17.551;
   1:  PR[91,3] = PR[90,3] + 89.885;
   1:L PR[91] R[100]mm/sec CNT100;
   1:  PR[91,1] = PR[90,1] + -48.527;
   1:  PR[91,2] = PR[90,2] + 16.958;
   1:  PR[91,3] = PR[90,3] + 89.891;
   1:L PR[91] R[100]mm/sec CNT100;
   1:  PR[91] = PR[90];
   1:  PR[91,1] = PR[90,1] + -51.523;
   1:  PR[91,2] = PR[90,2] + 13.631;
   1:  PR[91,3] = PR[90,3] + 91.195;
   1:L PR[91] R[100]mm/sec CNT100;
   1:  PR[91,1] = PR[90,1] + -53.566;
   1:  PR[91,2] = PR[90,2] + 11.379;
   1:  PR[91,3] = PR[90,3] + 89.919;
   1:L PR[91] R[100]mm/sec CNT100;
   1:  PR[91,1] = PR[90,1] + -55.500;
   1:  PR[91,2] = PR[90,2] + 9.146;
   1:  PR[91,3] = PR[90,3] + 89.932;
   1:L PR[91] R[100]mm/sec CNT100;
   1:  PR[91,1] = PR[90,1] + -57.602;
   1:  PR[91,2] = PR[90,2] + 5.064;
   1:  PR[91,3] = PR[90,3] + 89.945;
   1:L PR[91] R[100]mm/sec CNT100;
   1:  PR[91,1] = PR[90,1] + -57.980;
   1:  PR[91,2] = PR[90,2] + 4.293;
   1:  PR[91,3] = PR[90,3] + 89.965;
   1:L PR[91] R[100]mm/sec CNT100;
   1:  PR[91,1] = PR[90,1] + -58.798;
   1:  PR[91,2] = PR[90,2] + -0.549;
   1:  PR[91,3] = PR[90,3] + 89.969;
   1:L PR[91] R[100]mm/sec CNT100;
   1:  PR[91,1] = PR[90,1] + -58.839;
   1:  PR[91,2] = PR[90,2] + -0.745;
   1:  PR[91,3] = PR[90,3] + 89.990;
   1:L PR[91] R[100]mm/sec CNT100;
   1:  PR[91,1] = PR[90,1] + -58.330;
   1:  PR[91,2] = PR[90,2] + -3.391;
   1:  PR[91,3] = PR[90,3] + 89.991;
   1:L PR[91] R[100]mm/sec CNT100;
   1:  PR[91,1] = PR[90,1] + -58.204;
   1:  PR[91,2] = PR[90,2] + -3.732;
   1:  PR[91,3] = PR[90,3] + 90.003;
   1:L PR[91] R[100]mm/sec CNT100;
   1:  PR[91,1] = PR[90,1] + -57.931;
   1:  PR[91,2] = PR[90,2] + -5.477;
   1:  PR[91,3] = PR[90,3] + 90.004;
   1:L PR[91] R[100]mm/sec CNT100;
   1:  PR[91,1] = PR[90,1] + -56.698;
   1:  PR[91,2] = PR[90,2] + -8.113;
   1:  PR[91,3] = PR[90,3] + 90.012;
   1:L PR[91] R[100]mm/sec CNT100;
   1:  PR[91,1] = PR[90,1] + -55.683;
   1:  PR[91,2] = PR[90,2] + -10.216;
   1:  PR[91,3] = PR[90,3] + 90.025;
   1:L PR[91] R[100]mm/sec CNT100;
   1:  PR[91,1] = PR[90,1] + -54.260;
   1:  PR[91,2] = PR[90,2] + -11.952;
   1:  PR[91,3] = PR[90,3] + 90.035;
   1:L PR[91] R[100]mm/sec CNT100;
   1:  PR[91,1] = PR[90,1] + -51.781;
   1:  PR[91,2] = PR[90,2] + -14.870;
   1:  PR[91,3] = PR[90,3] + 90.045;
   1:L PR[91] R[100]mm/sec CNT100;
   1:  PR[91,1] = PR[90,1] + -51.015;
   1:  PR[91,2] = PR[90,2] + -15.487;
   1:  PR[91,3] = PR[90,3] + 90.061;
   1:L PR[91] R[100]mm/sec CNT100;
   1:  PR[91,1] = PR[90,1] + -48.599;
   1:  PR[91,2] = PR[90,2] + -17.345;
   1:  PR[91,3] = PR[90,3] + 90.066;
   1:L PR[91] R[100]mm/sec CNT100;
   1:  PR[91,1] = PR[90,1] + -46.209;
   1:  PR[91,2] = PR[90,2] + -18.944;
   1:  PR[91,3] = PR[90,3] + 90.079;
   1:L PR[91] R[100]mm/sec CNT100;
   1:  PR[91,1] = PR[90,1] + -44.861;
   1:  PR[91,2] = PR[90,2] + -19.639;
   1:  PR[91,3] = PR[90,3] + 90.092;
   1:L PR[91] R[100]mm/sec CNT100;
   1:  PR[91,1] = PR[90,1] + -40.414;
   1:  PR[91,2] = PR[90,2] + -21.682;
   1:  PR[91,3] = PR[90,3] + 90.098;
   1:L PR[91] R[100]mm/sec CNT100;
   1:  PR[91,1] = PR[90,1] + -35.551;
   1:  PR[91,2] = PR[90,2] + -23.564;
   1:  PR[91,3] = PR[90,3] + 90.119;
   1:L PR[91] R[100]mm/sec CNT100;
   1:  PR[91,1] = PR[90,1] + -27.190;
   1:  PR[91,2] = PR[90,2] + -25.737;
   1:  PR[91,3] = PR[90,3] + 90.142;
   1:L PR[91] R[100]mm/sec CNT100;
   1:  PR[91,1] = PR[90,1] + -17.967;
   1:  PR[91,2] = PR[90,2] + -27.391;
   1:  PR[91,3] = PR[90,3] + 90.180;
   1:L PR[91] R[100]mm/sec CNT100;
   1:  PR[91,1] = PR[90,1] + -12.621;
   1:  PR[91,2] = PR[90,2] + -27.975;
   1:  PR[91,3] = PR[90,3] + 90.221;
   1:L PR[91] R[100]mm/sec CNT100;
   1:  PR[91,1] = PR[90,1] + -8.086;
   1:  PR[91,2] = PR[90,2] + -28.448;
   1:  PR[91,3] = PR[90,3] + 90.244;
   1:L PR[91] R[100]mm/sec CNT100;
   1:  PR[91,1] = PR[90,1] + 2.289;
   1:  PR[91,2] = PR[90,2] + -28.838;
   1:  PR[91,3] = PR[90,3] + 90.264;
   1:L PR[91] R[100]mm/sec CNT100;
   1:  PR[91,1] = PR[90,1] + 10.823;
   1:  PR[91,2] = PR[90,2] + -28.561;
   1:  PR[91,3] = PR[90,3] + 90.309;
   1:L PR[91] R[100]mm/sec CNT100;
   1:  PR[91,1] = PR[90,1] + 13.810;
   1:  PR[91,2] = PR[90,2] + -28.429;
   1:  PR[91,3] = PR[90,3] + 90.347;
   1:L PR[91] R[100]mm/sec CNT100;
   1:  PR[91,1] = PR[90,1] + 15.592;
   1:  PR[91,2] = PR[90,2] + -28.281;
   1:  PR[91,3] = PR[90,3] + 90.360;
   1:L PR[91] R[100]mm/sec CNT100;
   1:  PR[91,1] = PR[90,1] + 18.160;
   1:  PR[91,2] = PR[90,2] + -28.542;
   1:  PR[91,3] = PR[90,3] + 90.367;
   1:L PR[91] R[100]mm/sec CNT100;
   1:  PR[91,1] = PR[90,1] + 19.296;
   1:  PR[91,2] = PR[90,2] + -28.595;
   1:  PR[91,3] = PR[90,3] + 90.379;
   1:L PR[91] R[100]mm/sec CNT100;
   1:  PR[91,1] = PR[90,1] + 23.157;
   1:  PR[91,2] = PR[90,2] + -28.523;
   1:  PR[91,3] = PR[90,3] + 90.384;
   1:L PR[91] R[100]mm/sec CNT100;
   1:  PR[91,1] = PR[90,1] + 23.238;
   1:  PR[91,2] = PR[90,2] + -28.935;
   1:  PR[91,3] = PR[90,3] + 90.400;
   1:L PR[91] R[100]mm/sec CNT100;
   1:  PR[91,1] = PR[90,1] + 27.173;
   1:  PR[91,2] = PR[90,2] + -29.863;
   1:  PR[91,3] = PR[90,3] + 90.402;
   1:L PR[91] R[100]mm/sec CNT100;
   1:  PR[91,1] = PR[90,1] + 32.444;
   1:  PR[91,2] = PR[90,2] + -30.151;
   1:  PR[91,3] = PR[90,3] + 90.420;
   1:L PR[91] R[100]mm/sec CNT100;
   1:  PR[91,1] = PR[90,1] + 37.636;
   1:  PR[91,2] = PR[90,2] + -29.526;
   1:  PR[91,3] = PR[90,3] + 90.443;
   1:L PR[91] R[100]mm/sec CNT100;
   1:  PR[91,1] = PR[90,1] + 42.574;
   1:  PR[91,2] = PR[90,2] + -28.024;
   1:  PR[91,3] = PR[90,3] + 90.466;
   1:L PR[91] R[100]mm/sec CNT100;
   1:  PR[91,1] = PR[90,1] + 47.097;
   1:  PR[91,2] = PR[90,2] + -25.706;
   1:  PR[91,3] = PR[90,3] + 90.488;
   1:L PR[91] R[100]mm/sec CNT100;
   1:  PR[91,1] = PR[90,1] + 48.892;
   1:  PR[91,2] = PR[90,2] + -24.337;
   1:  PR[91,3] = PR[90,3] + 90.510;
   1:L PR[91] R[100]mm/sec CNT100;
   1:  PR[91,1] = PR[90,1] + 51.223;
   1:  PR[91,2] = PR[90,2] + -22.665;
   1:  PR[91,3] = PR[90,3] + 90.520;
   1:L PR[91] R[100]mm/sec CNT100;
   1:  PR[91,1] = PR[90,1] + 54.732;
   1:  PR[91,2] = PR[90,2] + -19.081;
   1:  PR[91,3] = PR[90,3] + 90.533;
   1:L PR[91] R[100]mm/sec CNT100;
   1:  PR[91,1] = PR[90,1] + 57.517;
   1:  PR[91,2] = PR[90,2] + -14.985;
   1:  PR[91,3] = PR[90,3] + 90.555;
   1:L PR[91] R[100]mm/sec CNT100;
   1:  PR[91,1] = PR[90,1] + 58.305;
   1:  PR[91,2] = PR[90,2] + -13.230;
   1:  PR[91,3] = PR[90,3] + 90.576;
   1:L PR[91] R[100]mm/sec CNT100;
   1:  PR[91,1] = PR[90,1] + 59.505;
   1:  PR[91,2] = PR[90,2] + -10.878;
   1:  PR[91,3] = PR[90,3] + 90.585;
   1:L PR[91] R[100]mm/sec CNT100;
   1:  PR[91,1] = PR[90,1] + 59.774;
   1:  PR[91,2] = PR[90,2] + -10.289;
   1:  PR[91,3] = PR[90,3] + 90.596;
   1:L PR[91] R[100]mm/sec CNT100;
   1:  PR[91,1] = PR[90,1] + 60.701;
   1:  PR[91,2] = PR[90,2] + -7.100;
   1:  PR[91,3] = PR[90,3] + 90.599;
   1:L PR[91] R[100]mm/sec CNT100;
   1:  PR[91,1] = PR[90,1] + 61.119;
   1:  PR[91,2] = PR[90,2] + -5.502;
   1:  PR[91,3] = PR[90,3] + 90.613;
   1:L PR[91] R[100]mm/sec CNT100;
   1:  PR[91,1] = PR[90,1] + 61.319;
   1:  PR[91,2] = PR[90,2] + -3.222;
   1:  PR[91,3] = PR[90,3] + 90.621;
   1:L PR[91] R[100]mm/sec CNT100;
   1:  PR[91,1] = PR[90,1] + 61.346;
   1:  PR[91,2] = PR[90,2] + -2.444;
   1:  PR[91,3] = PR[90,3] + 90.631;
   1:L PR[91] R[100]mm/sec CNT100;
   1:  PR[91,1] = PR[90,1] + 61.506;
   1:  PR[91,2] = PR[90,2] + -0.705;
   1:  PR[91,3] = PR[90,3] + 90.634;
   1:L PR[91] R[100]mm/sec CNT100;
   1:  PR[91,1] = PR[90,1] + 61.354;
   1:  PR[91,2] = PR[90,2] + 1.542;
   1:  PR[91,3] = PR[90,3] + 90.642;
   1:L PR[91] R[100]mm/sec CNT100;
   1:  PR[91,1] = PR[90,1] + 61.121;
   1:  PR[91,2] = PR[90,2] + 4.037;
   1:  PR[91,3] = PR[90,3] + 90.651;
   1:L PR[91] R[100]mm/sec CNT100;
   1:  PR[91,1] = PR[90,1] + 60.700;
   1:  PR[91,2] = PR[90,2] + 5.641;
   1:  PR[91,3] = PR[90,3] + 90.662;
   1:L PR[91] R[100]mm/sec CNT100;
   1:  PR[91,1] = PR[90,1] + 59.774;
   1:  PR[91,2] = PR[90,2] + 8.830;
   1:  PR[91,3] = PR[90,3] + 90.670;
   1:L PR[91] R[100]mm/sec CNT100;
   1:  PR[91,1] = PR[90,1] + 59.505;
   1:  PR[91,2] = PR[90,2] + 9.420;
   1:  PR[91,3] = PR[90,3] + 90.684;
   1:L PR[91] R[100]mm/sec CNT100;
   1:  PR[91,1] = PR[90,1] + 58.305;
   1:  PR[91,2] = PR[90,2] + 11.771;
   1:  PR[91,3] = PR[90,3] + 90.687;
   1:L PR[91] R[100]mm/sec CNT100;
   1:  PR[91,1] = PR[90,1] + 57.517;
   1:  PR[91,2] = PR[90,2] + 13.526;
   1:  PR[91,3] = PR[90,3] + 90.698;
   1:L PR[91] R[100]mm/sec CNT100;
   1:  PR[91,1] = PR[90,1] + 54.732;
   1:  PR[91,2] = PR[90,2] + 17.622;
   1:  PR[91,3] = PR[90,3] + 90.707;
   1:L PR[91] R[100]mm/sec CNT100;
   1:  PR[91,1] = PR[90,1] + 51.223;
   1:  PR[91,2] = PR[90,2] + 21.207;
   1:  PR[91,3] = PR[90,3] + 90.728;
   1:L PR[91] R[100]mm/sec CNT100;
   1:  PR[91,1] = PR[90,1] + 48.892;
   1:  PR[91,2] = PR[90,2] + 22.879;
   1:  PR[91,3] = PR[90,3] + 90.750;
   1:L PR[91] R[100]mm/sec CNT100;
   1:  PR[91,1] = PR[90,1] + 47.097;
   1:  PR[91,2] = PR[90,2] + 24.247;
   1:  PR[91,3] = PR[90,3] + 90.763;
   1:L PR[91] R[100]mm/sec CNT100;
   1:  PR[91,1] = PR[90,1] + 42.574;
   1:  PR[91,2] = PR[90,2] + 26.566;
   1:  PR[91,3] = PR[90,3] + 90.773;
   1:L PR[91] R[100]mm/sec CNT100;
   1:  PR[91,1] = PR[90,1] + 37.636;
   1:  PR[91,2] = PR[90,2] + 28.067;
   1:  PR[91,3] = PR[90,3] + 90.795;
   1:L PR[91] R[100]mm/sec CNT100;
   1:  PR[91,1] = PR[90,1] + 32.444;
   1:  PR[91,2] = PR[90,2] + 28.693;
   1:  PR[91,3] = PR[90,3] + 90.817;
   1:L PR[91] R[100]mm/sec CNT100;
   1:  PR[91,1] = PR[90,1] + 27.173;
   1:  PR[91,2] = PR[90,2] + 28.404;
   1:  PR[91,3] = PR[90,3] + 90.840;
   1:L PR[91] R[100]mm/sec CNT100;
   1:  PR[91,1] = PR[90,1] + 21.692;
   1:  PR[91,2] = PR[90,2] + 27.112;
   1:  PR[91,3] = PR[90,3] + 90.863;
   1:L PR[91] R[100]mm/sec CNT100;
   1:  PR[91,1] = PR[90,1] + 19.306;
   1:  PR[91,2] = PR[90,2] + 27.137;
   1:  PR[91,3] = PR[90,3] + 90.888;
   1:L PR[91] R[100]mm/sec CNT100;
   1:  PR[91,1] = PR[90,1] + 18.181;
   1:  PR[91,2] = PR[90,2] + 27.085;
   1:  PR[91,3] = PR[90,3] + 90.898;
   1:L PR[91] R[100]mm/sec CNT100;
   1:  PR[91,1] = PR[90,1] + 16.551;
   1:  PR[91,2] = PR[90,2] + 26.885;
   1:  PR[91,3] = PR[90,3] + 90.903;
   1:L PR[91] R[100]mm/sec CNT100;
   1:  PR[91,1] = PR[90,1] + 15.549;
   1:  PR[91,2] = PR[90,2] + 26.826;
   1:  PR[91,3] = PR[90,3] + 90.910;
   1:L PR[91] R[100]mm/sec CNT100;
   1:  PR[91,1] = PR[90,1] + 13.803;
   1:  PR[91,2] = PR[90,2] + 26.970;
   1:  PR[91,3] = PR[90,3] + 90.914;
   1:L PR[91] R[100]mm/sec CNT100;
   1:  PR[91,1] = PR[90,1] + 12.939;
   1:  PR[91,2] = PR[90,2] + 27.013;
   1:  PR[91,3] = PR[90,3] + 90.922;
   1:L PR[91] R[100]mm/sec CNT100;
   1:  PR[91,1] = PR[90,1] + 8.683;
   1:  PR[91,2] = PR[90,2] + 27.178;
   1:  PR[91,3] = PR[90,3] + 90.926;
   1:L PR[91] R[100]mm/sec CNT100;
   1:  PR[91,1] = PR[90,1] + 2.290;
   1:  PR[91,2] = PR[90,2] + 27.379;
   1:  PR[91,3] = PR[90,3] + 90.944;
   1:L PR[91] R[100]mm/sec CNT100;
   1:  PR[91,1] = PR[90,1] + -8.086;
   1:  PR[91,2] = PR[90,2] + 26.989;
   1:  PR[91,3] = PR[90,3] + 90.972;
   1:L PR[91] R[100]mm/sec CNT100;
   1:  PR[91,1] = PR[90,1] + -12.621;
   1:  PR[91,2] = PR[90,2] + 26.516;
   1:  PR[91,3] = PR[90,3] + 91.018;
   1:L PR[91] R[100]mm/sec CNT100;
   1:  PR[91,1] = PR[90,1] + -17.967;
   1:  PR[91,2] = PR[90,2] + 25.932;
   1:  PR[91,3] = PR[90,3] + 91.037;
   1:L PR[91] R[100]mm/sec CNT100;
   1:  PR[91,1] = PR[90,1] + -27.190;
   1:  PR[91,2] = PR[90,2] + 24.278;
   1:  PR[91,3] = PR[90,3] + 91.061;
   1:L PR[91] R[100]mm/sec CNT100;
   1:  PR[91,1] = PR[90,1] + -35.555;
   1:  PR[91,2] = PR[90,2] + 22.104;
   1:  PR[91,3] = PR[90,3] + 91.102;
   1:L PR[91] R[100]mm/sec CNT100;
   1:  PR[91,1] = PR[90,1] + -40.381;
   1:  PR[91,2] = PR[90,2] + 20.261;
   1:  PR[91,3] = PR[90,3] + 91.139;
   1:L PR[91] R[100]mm/sec CNT100;
   1:  PR[91,1] = PR[90,1] + -45.678;
   1:  PR[91,2] = PR[90,2] + 17.818;
   1:  PR[91,3] = PR[90,3] + 91.162;
   1:L PR[91] R[100]mm/sec CNT100;
   1:  PR[91,1] = PR[90,1] + -46.273;
   1:  PR[91,2] = PR[90,2] + 17.514;
   1:  PR[91,3] = PR[90,3] + 91.187;
   1:L PR[91] R[100]mm/sec CNT100;
   1:  PR[91,1] = PR[90,1] + -47.159;
   1:  PR[91,2] = PR[90,2] + 16.922;
   1:  PR[91,3] = PR[90,3] + 91.190;
   1:L PR[91] R[100]mm/sec CNT100;
   1:  PR[91] = PR[90];
   1:  PR[91,1] = PR[90,1] + -50.121;
   1:  PR[91,2] = PR[90,2] + 13.621;
   1:  PR[91,3] = PR[90,3] + 92.495;
   1:L PR[91] R[100]mm/sec CNT100;
   1:  PR[91,1] = PR[90,1] + -51.090;
   1:  PR[91,2] = PR[90,2] + 12.553;
   1:  PR[91,3] = PR[90,3] + 91.207;
   1:L PR[91] R[100]mm/sec CNT100;
   1:  PR[91,1] = PR[90,1] + -54.051;
   1:  PR[91,2] = PR[90,2] + 9.133;
   1:  PR[91,3] = PR[90,3] + 91.213;
   1:L PR[91] R[100]mm/sec CNT100;
   1:  PR[91,1] = PR[90,1] + -55.580;
   1:  PR[91,2] = PR[90,2] + 6.165;
   1:  PR[91,3] = PR[90,3] + 91.233;
   1:L PR[91] R[100]mm/sec CNT100;
   1:  PR[91,1] = PR[90,1] + -56.502;
   1:  PR[91,2] = PR[90,2] + 4.285;
   1:  PR[91,3] = PR[90,3] + 91.248;
   1:L PR[91] R[100]mm/sec CNT100;
   1:  PR[91,1] = PR[90,1] + -57.148;
   1:  PR[91,2] = PR[90,2] + 0.460;
   1:  PR[91,3] = PR[90,3] + 91.257;
   1:L PR[91] R[100]mm/sec CNT100;
   1:  PR[91,1] = PR[90,1] + -57.399;
   1:  PR[91,2] = PR[90,2] + -0.745;
   1:  PR[91,3] = PR[90,3] + 91.274;
   1:L PR[91] R[100]mm/sec CNT100;
   1:  PR[91,1] = PR[90,1] + -57.058;
   1:  PR[91,2] = PR[90,2] + -2.522;
   1:  PR[91,3] = PR[90,3] + 91.279;
   1:L PR[91] R[100]mm/sec CNT100;
   1:  PR[91,1] = PR[90,1] + -56.883;
   1:  PR[91,2] = PR[90,2] + -2.998;
   1:  PR[91,3] = PR[90,3] + 91.287;
   1:L PR[91] R[100]mm/sec CNT100;
   1:  PR[91,1] = PR[90,1] + -56.485;
   1:  PR[91,2] = PR[90,2] + -5.538;
   1:  PR[91,3] = PR[90,3] + 91.290;
   1:L PR[91] R[100]mm/sec CNT100;
   1:  PR[91,1] = PR[90,1] + -55.562;
   1:  PR[91,2] = PR[90,2] + -7.510;
   1:  PR[91,3] = PR[90,3] + 91.301;
   1:L PR[91] R[100]mm/sec CNT100;
   1:  PR[91,1] = PR[90,1] + -54.199;
   1:  PR[91,2] = PR[90,2] + -10.337;
   1:  PR[91,3] = PR[90,3] + 91.311;
   1:L PR[91] R[100]mm/sec CNT100;
   1:  PR[91,1] = PR[90,1] + -53.264;
   1:  PR[91,2] = PR[90,2] + -11.477;
   1:  PR[91,3] = PR[90,3] + 91.324;
   1:L PR[91] R[100]mm/sec CNT100;
   1:  PR[91,1] = PR[90,1] + -50.242;
   1:  PR[91,2] = PR[90,2] + -15.034;
   1:  PR[91,3] = PR[90,3] + 91.331;
   1:L PR[91] R[100]mm/sec CNT100;
   1:  PR[91,1] = PR[90,1] + -49.453;
   1:  PR[91,2] = PR[90,2] + -15.648;
   1:  PR[91,3] = PR[90,3] + 91.351;
   1:L PR[91] R[100]mm/sec CNT100;
   1:  PR[91,1] = PR[90,1] + -44.605;
   1:  PR[91,2] = PR[90,2] + -18.891;
   1:  PR[91,3] = PR[90,3] + 91.356;
   1:L PR[91] R[100]mm/sec CNT100;
   1:  PR[91,1] = PR[90,1] + -41.813;
   1:  PR[91,2] = PR[90,2] + -20.331;
   1:  PR[91,3] = PR[90,3] + 91.382;
   1:L PR[91] R[100]mm/sec CNT100;
   1:  PR[91,1] = PR[90,1] + -39.127;
   1:  PR[91,2] = PR[90,2] + -21.566;
   1:  PR[91,3] = PR[90,3] + 91.395;
   1:L PR[91] R[100]mm/sec CNT100;
   1:  PR[91,1] = PR[90,1] + -36.152;
   1:  PR[91,2] = PR[90,2] + -22.717;
   1:  PR[91,3] = PR[90,3] + 91.408;
   1:L PR[91] R[100]mm/sec CNT100;
   1:  PR[91,1] = PR[90,1] + -33.238;
   1:  PR[91,2] = PR[90,2] + -23.753;
   1:  PR[91,3] = PR[90,3] + 91.423;
   1:L PR[91] R[100]mm/sec CNT100;
   1:  PR[91,1] = PR[90,1] + -24.786;
   1:  PR[91,2] = PR[90,2] + -25.953;
   1:  PR[91,3] = PR[90,3] + 91.436;
   1:L PR[91] R[100]mm/sec CNT100;
   1:  PR[91,1] = PR[90,1] + -21.549;
   1:  PR[91,2] = PR[90,2] + -26.545;
   1:  PR[91,3] = PR[90,3] + 91.475;
   1:L PR[91] R[100]mm/sec CNT100;
   1:  PR[91,1] = PR[90,1] + -15.498;
   1:  PR[91,2] = PR[90,2] + -27.623;
   1:  PR[91,3] = PR[90,3] + 91.489;
   1:L PR[91] R[100]mm/sec CNT100;
   1:  PR[91,1] = PR[90,1] + -9.208;
   1:  PR[91,2] = PR[90,2] + -28.310;
   1:  PR[91,3] = PR[90,3] + 91.516;
   1:L PR[91] R[100]mm/sec CNT100;
   1:  PR[91,1] = PR[90,1] + -5.540;
   1:  PR[91,2] = PR[90,2] + -28.692;
   1:  PR[91,3] = PR[90,3] + 91.544;
   1:L PR[91] R[100]mm/sec CNT100;
   1:  PR[91,1] = PR[90,1] + 4.915;
   1:  PR[91,2] = PR[90,2] + -29.090;
   1:  PR[91,3] = PR[90,3] + 91.560;
   1:L PR[91] R[100]mm/sec CNT100;
   1:  PR[91,1] = PR[90,1] + 11.842;
   1:  PR[91,2] = PR[90,2] + -28.857;
   1:  PR[91,3] = PR[90,3] + 91.606;
   1:L PR[91] R[100]mm/sec CNT100;
   1:  PR[91,1] = PR[90,1] + 16.065;
   1:  PR[91,2] = PR[90,2] + -28.677;
   1:  PR[91,3] = PR[90,3] + 91.637;
   1:L PR[91] R[100]mm/sec CNT100;
   1:  PR[91,1] = PR[90,1] + 17.327;
   1:  PR[91,2] = PR[90,2] + -28.590;
   1:  PR[91,3] = PR[90,3] + 91.656;
   1:L PR[91] R[100]mm/sec CNT100;
   1:  PR[91,1] = PR[90,1] + 18.267;
   1:  PR[91,2] = PR[90,2] + -28.686;
   1:  PR[91,3] = PR[90,3] + 91.661;
   1:L PR[91] R[100]mm/sec CNT100;
   1:  PR[91,1] = PR[90,1] + 19.931;
   1:  PR[91,2] = PR[90,2] + -28.763;
   1:  PR[91,3] = PR[90,3] + 91.665;
   1:L PR[91] R[100]mm/sec CNT100;
   1:  PR[91,1] = PR[90,1] + 22.994;
   1:  PR[91,2] = PR[90,2] + -28.705;
   1:  PR[91,3] = PR[90,3] + 91.673;
   1:L PR[91] R[100]mm/sec CNT100;
   1:  PR[91,1] = PR[90,1] + 23.074;
   1:  PR[91,2] = PR[90,2] + -29.110;
   1:  PR[91,3] = PR[90,3] + 91.686;
   1:L PR[91] R[100]mm/sec CNT100;
   1:  PR[91,1] = PR[90,1] + 26.769;
   1:  PR[91,2] = PR[90,2] + -29.990;
   1:  PR[91,3] = PR[90,3] + 91.688;
   1:L PR[91] R[100]mm/sec CNT100;
   1:  PR[91,1] = PR[90,1] + 27.259;
   1:  PR[91,2] = PR[90,2] + -30.069;
   1:  PR[91,3] = PR[90,3] + 91.705;
   1:L PR[91] R[100]mm/sec CNT100;
   1:  PR[91,1] = PR[90,1] + 32.225;
   1:  PR[91,2] = PR[90,2] + -30.343;
   1:  PR[91,3] = PR[90,3] + 91.707;
   1:L PR[91] R[100]mm/sec CNT100;
   1:  PR[91,1] = PR[90,1] + 37.453;
   1:  PR[91,2] = PR[90,2] + -29.713;
   1:  PR[91,3] = PR[90,3] + 91.729;
   1:L PR[91] R[100]mm/sec CNT100;
   1:  PR[91,1] = PR[90,1] + 42.429;
   1:  PR[91,2] = PR[90,2] + -28.207;
   1:  PR[91,3] = PR[90,3] + 91.752;
   1:L PR[91] R[100]mm/sec CNT100;
   1:  PR[91,1] = PR[90,1] + 44.848;
   1:  PR[91,2] = PR[90,2] + -26.963;
   1:  PR[91,3] = PR[90,3] + 91.775;
   1:L PR[91] R[100]mm/sec CNT100;
   1:  PR[91,1] = PR[90,1] + 47.005;
   1:  PR[91,2] = PR[90,2] + -25.877;
   1:  PR[91,3] = PR[90,3] + 91.787;
   1:L PR[91] R[100]mm/sec CNT100;
   1:  PR[91,1] = PR[90,1] + 51.024;
   1:  PR[91,2] = PR[90,2] + -22.820;
   1:  PR[91,3] = PR[90,3] + 91.798;
   1:L PR[91] R[100]mm/sec CNT100;
   1:  PR[91,1] = PR[90,1] + 52.149;
   1:  PR[91,2] = PR[90,2] + -21.599;
   1:  PR[91,3] = PR[90,3] + 91.820;
   1:L PR[91] R[100]mm/sec CNT100;
   1:  PR[91,1] = PR[90,1] + 54.553;
   1:  PR[91,2] = PR[90,2] + -19.145;
   1:  PR[91,3] = PR[90,3] + 91.827;
   1:L PR[91] R[100]mm/sec CNT100;
   1:  PR[91,1] = PR[90,1] + 57.366;
   1:  PR[91,2] = PR[90,2] + -15.027;
   1:  PR[91,3] = PR[90,3] + 91.842;
   1:L PR[91] R[100]mm/sec CNT100;
   1:  PR[91,1] = PR[90,1] + 59.402;
   1:  PR[91,2] = PR[90,2] + -10.505;
   1:  PR[91,3] = PR[90,3] + 91.864;
   1:L PR[91] R[100]mm/sec CNT100;
   1:  PR[91,1] = PR[90,1] + 60.496;
   1:  PR[91,2] = PR[90,2] + -6.223;
   1:  PR[91,3] = PR[90,3] + 91.886;
   1:L PR[91] R[100]mm/sec CNT100;
   1:  PR[91,1] = PR[90,1] + 60.661;
   1:  PR[91,2] = PR[90,2] + -5.644;
   1:  PR[91,3] = PR[90,3] + 91.906;
   1:L PR[91] R[100]mm/sec CNT100;
   1:  PR[91,1] = PR[90,1] + 61.112;
   1:  PR[91,2] = PR[90,2] + -0.706;
   1:  PR[91,3] = PR[90,3] + 91.908;
   1:L PR[91] R[100]mm/sec CNT100;
   1:  PR[91,1] = PR[90,1] + 61.095;
   1:  PR[91,2] = PR[90,2] + -0.444;
   1:  PR[91,3] = PR[90,3] + 91.930;
   1:L PR[91] R[100]mm/sec CNT100;
   1:  PR[91,1] = PR[90,1] + 60.662;
   1:  PR[91,2] = PR[90,2] + 4.183;
   1:  PR[91,3] = PR[90,3] + 91.931;
   1:L PR[91] R[100]mm/sec CNT100;
   1:  PR[91,1] = PR[90,1] + 60.496;
   1:  PR[91,2] = PR[90,2] + 4.764;
   1:  PR[91,3] = PR[90,3] + 91.952;
   1:L PR[91] R[100]mm/sec CNT100;
   1:  PR[91,1] = PR[90,1] + 59.402;
   1:  PR[91,2] = PR[90,2] + 9.046;
   1:  PR[91,3] = PR[90,3] + 91.954;
   1:L PR[91] R[100]mm/sec CNT100;
   1:  PR[91,1] = PR[90,1] + 57.365;
   1:  PR[91,2] = PR[90,2] + 13.568;
   1:  PR[91,3] = PR[90,3] + 91.974;
   1:L PR[91] R[100]mm/sec CNT100;
   1:  PR[91,1] = PR[90,1] + 54.553;
   1:  PR[91,2] = PR[90,2] + 17.686;
   1:  PR[91,3] = PR[90,3] + 91.996;
   1:L PR[91] R[100]mm/sec CNT100;
   1:  PR[91,1] = PR[90,1] + 52.149;
   1:  PR[91,2] = PR[90,2] + 20.140;
   1:  PR[91,3] = PR[90,3] + 92.018;
   1:L PR[91] R[100]mm/sec CNT100;
   1:  PR[91,1] = PR[90,1] + 51.024;
   1:  PR[91,2] = PR[90,2] + 21.361;
   1:  PR[91,3] = PR[90,3] + 92.033;
   1:L PR[91] R[100]mm/sec CNT100;
   1:  PR[91,1] = PR[90,1] + 47.005;
   1:  PR[91,2] = PR[90,2] + 24.418;
   1:  PR[91,3] = PR[90,3] + 92.040;
   1:L PR[91] R[100]mm/sec CNT100;
   1:  PR[91,1] = PR[90,1] + 44.848;
   1:  PR[91,2] = PR[90,2] + 25.504;
   1:  PR[91,3] = PR[90,3] + 92.062;
   1:L PR[91] R[100]mm/sec CNT100;
   1:  PR[91,1] = PR[90,1] + 42.429;
   1:  PR[91,2] = PR[90,2] + 26.748;
   1:  PR[91,3] = PR[90,3] + 92.073;
   1:L PR[91] R[100]mm/sec CNT100;
   1:  PR[91,1] = PR[90,1] + 37.453;
   1:  PR[91,2] = PR[90,2] + 28.254;
   1:  PR[91,3] = PR[90,3] + 92.085;
   1:L PR[91] R[100]mm/sec CNT100;
   1:  PR[91,1] = PR[90,1] + 32.225;
   1:  PR[91,2] = PR[90,2] + 28.884;
   1:  PR[91,3] = PR[90,3] + 92.108;
   1:L PR[91] R[100]mm/sec CNT100;
   1:  PR[91,1] = PR[90,1] + 27.261;
   1:  PR[91,2] = PR[90,2] + 28.611;
   1:  PR[91,3] = PR[90,3] + 92.131;
   1:L PR[91] R[100]mm/sec CNT100;
   1:  PR[91,1] = PR[90,1] + 26.766;
   1:  PR[91,2] = PR[90,2] + 28.530;
   1:  PR[91,3] = PR[90,3] + 92.153;
   1:L PR[91] R[100]mm/sec CNT100;
   1:  PR[91,1] = PR[90,1] + 21.551;
   1:  PR[91,2] = PR[90,2] + 27.288;
   1:  PR[91,3] = PR[90,3] + 92.155;
   1:L PR[91] R[100]mm/sec CNT100;
   1:  PR[91,1] = PR[90,1] + 19.940;
   1:  PR[91,2] = PR[90,2] + 27.304;
   1:  PR[91,3] = PR[90,3] + 92.179;
   1:L PR[91] R[100]mm/sec CNT100;
   1:  PR[91,1] = PR[90,1] + 18.289;
   1:  PR[91,2] = PR[90,2] + 27.228;
   1:  PR[91,3] = PR[90,3] + 92.186;
   1:L PR[91] R[100]mm/sec CNT100;
   1:  PR[91,1] = PR[90,1] + 17.745;
   1:  PR[91,2] = PR[90,2] + 27.162;
   1:  PR[91,3] = PR[90,3] + 92.193;
   1:L PR[91] R[100]mm/sec CNT100;
   1:  PR[91,1] = PR[90,1] + 17.271;
   1:  PR[91,2] = PR[90,2] + 27.133;
   1:  PR[91,3] = PR[90,3] + 92.196;
   1:L PR[91] R[100]mm/sec CNT100;
   1:  PR[91,1] = PR[90,1] + 16.605;
   1:  PR[91,2] = PR[90,2] + 27.189;
   1:  PR[91,3] = PR[90,3] + 92.198;
   1:L PR[91] R[100]mm/sec CNT100;
   1:  PR[91,1] = PR[90,1] + 15.610;
   1:  PR[91,2] = PR[90,2] + 27.240;
   1:  PR[91,3] = PR[90,3] + 92.201;
   1:L PR[91] R[100]mm/sec CNT100;
   1:  PR[91,1] = PR[90,1] + 8.035;
   1:  PR[91,2] = PR[90,2] + 27.533;
   1:  PR[91,3] = PR[90,3] + 92.205;
   1:L PR[91] R[100]mm/sec CNT100;
   1:  PR[91,1] = PR[90,1] + 4.917;
   1:  PR[91,2] = PR[90,2] + 27.632;
   1:  PR[91,3] = PR[90,3] + 92.239;
   1:L PR[91] R[100]mm/sec CNT100;
   1:  PR[91,1] = PR[90,1] + -5.540;
   1:  PR[91,2] = PR[90,2] + 27.233;
   1:  PR[91,3] = PR[90,3] + 92.252;
   1:L PR[91] R[100]mm/sec CNT100;
   1:  PR[91,1] = PR[90,1] + -9.208;
   1:  PR[91,2] = PR[90,2] + 26.851;
   1:  PR[91,3] = PR[90,3] + 92.298;
   1:L PR[91] R[100]mm/sec CNT100;
   1:  PR[91,1] = PR[90,1] + -15.498;
   1:  PR[91,2] = PR[90,2] + 26.164;
   1:  PR[91,3] = PR[90,3] + 92.315;
   1:L PR[91] R[100]mm/sec CNT100;
   1:  PR[91,1] = PR[90,1] + -21.549;
   1:  PR[91,2] = PR[90,2] + 25.086;
   1:  PR[91,3] = PR[90,3] + 92.343;
   1:L PR[91] R[100]mm/sec CNT100;
   1:  PR[91,1] = PR[90,1] + -24.786;
   1:  PR[91,2] = PR[90,2] + 24.494;
   1:  PR[91,3] = PR[90,3] + 92.370;
   1:L PR[91] R[100]mm/sec CNT100;
   1:  PR[91,1] = PR[90,1] + -33.238;
   1:  PR[91,2] = PR[90,2] + 22.294;
   1:  PR[91,3] = PR[90,3] + 92.384;
   1:L PR[91] R[100]mm/sec CNT100;
   1:  PR[91,1] = PR[90,1] + -36.156;
   1:  PR[91,2] = PR[90,2] + 21.257;
   1:  PR[91,3] = PR[90,3] + 92.423;
   1:L PR[91] R[100]mm/sec CNT100;
   1:  PR[91,1] = PR[90,1] + -39.108;
   1:  PR[91,2] = PR[90,2] + 20.129;
   1:  PR[91,3] = PR[90,3] + 92.436;
   1:L PR[91] R[100]mm/sec CNT100;
   1:  PR[91,1] = PR[90,1] + -42.315;
   1:  PR[91,2] = PR[90,2] + 18.650;
   1:  PR[91,3] = PR[90,3] + 92.450;
   1:L PR[91] R[100]mm/sec CNT100;
   1:  PR[91,1] = PR[90,1] + -44.657;
   1:  PR[91,2] = PR[90,2] + 17.456;
   1:  PR[91,3] = PR[90,3] + 92.466;
   1:L PR[91] R[100]mm/sec CNT100;
   1:  PR[91,1] = PR[90,1] + -47.997;
   1:  PR[91,2] = PR[90,2] + 15.223;
   1:  PR[91,3] = PR[90,3] + 92.477;
   1:L PR[91] R[100]mm/sec CNT100;
   1:  PR[91] = PR[90];
   1:  PR[91,1] = PR[90,1] + -52.602;
   1:  PR[91,2] = PR[90,2] + 9.120;
   1:  PR[91,3] = PR[90,3] + 93.795;
   1:L PR[91] R[100]mm/sec CNT100;
   1:  PR[91,1] = PR[90,1] + -53.557;
   1:  PR[91,2] = PR[90,2] + 7.266;
   1:  PR[91,3] = PR[90,3] + 92.521;
   1:L PR[91] R[100]mm/sec CNT100;
   1:  PR[91,1] = PR[90,1] + -55.024;
   1:  PR[91,2] = PR[90,2] + 4.276;
   1:  PR[91,3] = PR[90,3] + 92.531;
   1:L PR[91] R[100]mm/sec CNT100;
   1:  PR[91,1] = PR[90,1] + -55.498;
   1:  PR[91,2] = PR[90,2] + 1.469;
   1:  PR[91,3] = PR[90,3] + 92.545;
   1:L PR[91] R[100]mm/sec CNT100;
   1:  PR[91,1] = PR[90,1] + -55.960;
   1:  PR[91,2] = PR[90,2] + -0.745;
   1:  PR[91,3] = PR[90,3] + 92.558;
   1:L PR[91] R[100]mm/sec CNT100;
   1:  PR[91,1] = PR[90,1] + -55.785;
   1:  PR[91,2] = PR[90,2] + -1.653;
   1:  PR[91,3] = PR[90,3] + 92.568;
   1:L PR[91] R[100]mm/sec CNT100;
   1:  PR[91,1] = PR[90,1] + -55.561;
   1:  PR[91,2] = PR[90,2] + -2.263;
   1:  PR[91,3] = PR[90,3] + 92.572;
   1:L PR[91] R[100]mm/sec CNT100;
   1:  PR[91,1] = PR[90,1] + -55.038;
   1:  PR[91,2] = PR[90,2] + -5.599;
   1:  PR[91,3] = PR[90,3] + 92.575;
   1:L PR[91] R[100]mm/sec CNT100;
   1:  PR[91,1] = PR[90,1] + -54.426;
   1:  PR[91,2] = PR[90,2] + -6.908;
   1:  PR[91,3] = PR[90,3] + 92.590;
   1:L PR[91] R[100]mm/sec CNT100;
   1:  PR[91,1] = PR[90,1] + -52.715;
   1:  PR[91,2] = PR[90,2] + -10.457;
   1:  PR[91,3] = PR[90,3] + 92.597;
   1:L PR[91] R[100]mm/sec CNT100;
   1:  PR[91,1] = PR[90,1] + -52.268;
   1:  PR[91,2] = PR[90,2] + -11.002;
   1:  PR[91,3] = PR[90,3] + 92.614;
   1:L PR[91] R[100]mm/sec CNT100;
   1:  PR[91,1] = PR[90,1] + -50.009;
   1:  PR[91,2] = PR[90,2] + -13.661;
   1:  PR[91,3] = PR[90,3] + 92.617;
   1:L PR[91] R[100]mm/sec CNT100;
   1:  PR[91,1] = PR[90,1] + -48.814;
   1:  PR[91,2] = PR[90,2] + -14.872;
   1:  PR[91,3] = PR[90,3] + 92.633;
   1:L PR[91] R[100]mm/sec CNT100;
   1:  PR[91,1] = PR[90,1] + -48.612;
   1:  PR[91,2] = PR[90,2] + -15.066;
   1:  PR[91,3] = PR[90,3] + 92.640;
   1:L PR[91] R[100]mm/sec CNT100;
   1:  PR[91,1] = PR[90,1] + -47.915;
   1:  PR[91,2] = PR[90,2] + -15.552;
   1:  PR[91,3] = PR[90,3] + 92.642;
   1:L PR[91] R[100]mm/sec CNT100;
   1:  PR[91,1] = PR[90,1] + -43.001;
   1:  PR[91,2] = PR[90,2] + -18.839;
   1:  PR[91,3] = PR[90,3] + 92.645;
   1:L PR[91] R[100]mm/sec CNT100;
   1:  PR[91,1] = PR[90,1] + -38.766;
   1:  PR[91,2] = PR[90,2] + -21.024;
   1:  PR[91,3] = PR[90,3] + 92.672;
   1:L PR[91] R[100]mm/sec CNT100;
   1:  PR[91,1] = PR[90,1] + -37.840;
   1:  PR[91,2] = PR[90,2] + -21.449;
   1:  PR[91,3] = PR[90,3] + 92.693;
   1:L PR[91] R[100]mm/sec CNT100;
   1:  PR[91,1] = PR[90,1] + -36.800;
   1:  PR[91,2] = PR[90,2] + -21.851;
   1:  PR[91,3] = PR[90,3] + 92.698;
   1:L PR[91] R[100]mm/sec CNT100;
   1:  PR[91,1] = PR[90,1] + -30.899;
   1:  PR[91,2] = PR[90,2] + -23.948;
   1:  PR[91,3] = PR[90,3] + 92.702;
   1:L PR[91] R[100]mm/sec CNT100;
   1:  PR[91,1] = PR[90,1] + -22.384;
   1:  PR[91,2] = PR[90,2] + -26.169;
   1:  PR[91,3] = PR[90,3] + 92.730;
   1:L PR[91] R[100]mm/sec CNT100;
   1:  PR[91,1] = PR[90,1] + -18.279;
   1:  PR[91,2] = PR[90,2] + -26.920;
   1:  PR[91,3] = PR[90,3] + 92.770;
   1:L PR[91] R[100]mm/sec CNT100;
   1:  PR[91,1] = PR[90,1] + -13.027;
   1:  PR[91,2] = PR[90,2] + -27.855;
   1:  PR[91,3] = PR[90,3] + 92.788;
   1:L PR[91] R[100]mm/sec CNT100;
   1:  PR[91,1] = PR[90,1] + -5.796;
   1:  PR[91,2] = PR[90,2] + -28.645;
   1:  PR[91,3] = PR[90,3] + 92.812;
   1:L PR[91] R[100]mm/sec CNT100;
   1:  PR[91,1] = PR[90,1] + -2.993;
   1:  PR[91,2] = PR[90,2] + -28.937;
   1:  PR[91,3] = PR[90,3] + 92.844;
   1:L PR[91] R[100]mm/sec CNT100;
   1:  PR[91,1] = PR[90,1] + 7.528;
   1:  PR[91,2] = PR[90,2] + -29.343;
   1:  PR[91,3] = PR[90,3] + 92.857;
   1:L PR[91] R[100]mm/sec CNT100;
   1:  PR[91,1] = PR[90,1] + 12.860;
   1:  PR[91,2] = PR[90,2] + -29.154;
   1:  PR[91,3] = PR[90,3] + 92.904;
   1:L PR[91] R[100]mm/sec CNT100;
   1:  PR[91,1] = PR[90,1] + 18.504;
   1:  PR[91,2] = PR[90,2] + -28.915;
   1:  PR[91,3] = PR[90,3] + 92.927;
   1:L PR[91] R[100]mm/sec CNT100;
   1:  PR[91,1] = PR[90,1] + 19.231;
   1:  PR[91,2] = PR[90,2] + -28.869;
   1:  PR[91,3] = PR[90,3] + 92.952;
   1:L PR[91] R[100]mm/sec CNT100;
   1:  PR[91,1] = PR[90,1] + 20.565;
   1:  PR[91,2] = PR[90,2] + -28.931;
   1:  PR[91,3] = PR[90,3] + 92.956;
   1:L PR[91] R[100]mm/sec CNT100;
   1:  PR[91,1] = PR[90,1] + 22.832;
   1:  PR[91,2] = PR[90,2] + -28.888;
   1:  PR[91,3] = PR[90,3] + 92.962;
   1:L PR[91] R[100]mm/sec CNT100;
   1:  PR[91,1] = PR[90,1] + 22.910;
   1:  PR[91,2] = PR[90,2] + -29.281;
   1:  PR[91,3] = PR[90,3] + 92.972;
   1:L PR[91] R[100]mm/sec CNT100;
   1:  PR[91,1] = PR[90,1] + 26.167;
   1:  PR[91,2] = PR[90,2] + -30.059;
   1:  PR[91,3] = PR[90,3] + 92.974;
   1:L PR[91] R[100]mm/sec CNT100;
   1:  PR[91,1] = PR[90,1] + 27.564;
   1:  PR[91,2] = PR[90,2] + -30.285;
   1:  PR[91,3] = PR[90,3] + 92.988;
   1:L PR[91] R[100]mm/sec CNT100;
   1:  PR[91,1] = PR[90,1] + 31.764;
   1:  PR[91,2] = PR[90,2] + -30.517;
   1:  PR[91,3] = PR[90,3] + 92.995;
   1:L PR[91] R[100]mm/sec CNT100;
   1:  PR[91,1] = PR[90,1] + 32.510;
   1:  PR[91,2] = PR[90,2] + -30.502;
   1:  PR[91,3] = PR[90,3] + 93.013;
   1:L PR[91] R[100]mm/sec CNT100;
   1:  PR[91,1] = PR[90,1] + 37.245;
   1:  PR[91,2] = PR[90,2] + -29.906;
   1:  PR[91,3] = PR[90,3] + 93.017;
   1:L PR[91] R[100]mm/sec CNT100;
   1:  PR[91,1] = PR[90,1] + 42.292;
   1:  PR[91,2] = PR[90,2] + -28.387;
   1:  PR[91,3] = PR[90,3] + 93.038;
   1:L PR[91] R[100]mm/sec CNT100;
   1:  PR[91,1] = PR[90,1] + 46.902;
   1:  PR[91,2] = PR[90,2] + -26.054;
   1:  PR[91,3] = PR[90,3] + 93.061;
   1:L PR[91] R[100]mm/sec CNT100;
   1:  PR[91,1] = PR[90,1] + 49.030;
   1:  PR[91,2] = PR[90,2] + -24.431;
   1:  PR[91,3] = PR[90,3] + 93.084;
   1:L PR[91] R[100]mm/sec CNT100;
   1:  PR[91,1] = PR[90,1] + 50.984;
   1:  PR[91,2] = PR[90,2] + -22.977;
   1:  PR[91,3] = PR[90,3] + 93.096;
   1:L PR[91] R[100]mm/sec CNT100;
   1:  PR[91,1] = PR[90,1] + 54.397;
   1:  PR[91,2] = PR[90,2] + -19.283;
   1:  PR[91,3] = PR[90,3] + 93.107;
   1:L PR[91] R[100]mm/sec CNT100;
   1:  PR[91,1] = PR[90,1] + 55.453;
   1:  PR[91,2] = PR[90,2] + -17.640;
   1:  PR[91,3] = PR[90,3] + 93.130;
   1:L PR[91] R[100]mm/sec CNT100;
   1:  PR[91,1] = PR[90,1] + 57.214;
   1:  PR[91,2] = PR[90,2] + -15.068;
   1:  PR[91,3] = PR[90,3] + 93.138;
   1:L PR[91] R[100]mm/sec CNT100;
   1:  PR[91,1] = PR[90,1] + 59.274;
   1:  PR[91,2] = PR[90,2] + -10.527;
   1:  PR[91,3] = PR[90,3] + 93.152;
   1:L PR[91] R[100]mm/sec CNT100;
   1:  PR[91,1] = PR[90,1] + 60.517;
   1:  PR[91,2] = PR[90,2] + -5.701;
   1:  PR[91,3] = PR[90,3] + 93.174;
   1:L PR[91] R[100]mm/sec CNT100;
   1:  PR[91,1] = PR[90,1] + 60.793;
   1:  PR[91,2] = PR[90,2] + -2.425;
   1:  PR[91,3] = PR[90,3] + 93.197;
   1:L PR[91] R[100]mm/sec CNT100;
   1:  PR[91,1] = PR[90,1] + 60.883;
   1:  PR[91,2] = PR[90,2] + -0.761;
   1:  PR[91,3] = PR[90,3] + 93.211;
   1:L PR[91] R[100]mm/sec CNT100;
   1:  PR[91,1] = PR[90,1] + 60.748;
   1:  PR[91,2] = PR[90,2] + 0.799;
   1:  PR[91,3] = PR[90,3] + 93.219;
   1:L PR[91] R[100]mm/sec CNT100;
   1:  PR[91,1] = PR[90,1] + 60.667;
   1:  PR[91,2] = PR[90,2] + 2.423;
   1:  PR[91,3] = PR[90,3] + 93.226;
   1:L PR[91] R[100]mm/sec CNT100;
   1:  PR[91,1] = PR[90,1] + 60.517;
   1:  PR[91,2] = PR[90,2] + 4.243;
   1:  PR[91,3] = PR[90,3] + 93.233;
   1:L PR[91] R[100]mm/sec CNT100;
   1:  PR[91,1] = PR[90,1] + 59.274;
   1:  PR[91,2] = PR[90,2] + 9.068;
   1:  PR[91,3] = PR[90,3] + 93.241;
   1:L PR[91] R[100]mm/sec CNT100;
   1:  PR[91,1] = PR[90,1] + 57.214;
   1:  PR[91,2] = PR[90,2] + 13.609;
   1:  PR[91,3] = PR[90,3] + 93.263;
   1:L PR[91] R[100]mm/sec CNT100;
   1:  PR[91,1] = PR[90,1] + 55.453;
   1:  PR[91,2] = PR[90,2] + 16.181;
   1:  PR[91,3] = PR[90,3] + 93.285;
   1:L PR[91] R[100]mm/sec CNT100;
   1:  PR[91,1] = PR[90,1] + 54.397;
   1:  PR[91,2] = PR[90,2] + 17.825;
   1:  PR[91,3] = PR[90,3] + 93.299;
   1:L PR[91] R[100]mm/sec CNT100;
   1:  PR[91,1] = PR[90,1] + 50.984;
   1:  PR[91,2] = PR[90,2] + 21.518;
   1:  PR[91,3] = PR[90,3] + 93.308;
   1:L PR[91] R[100]mm/sec CNT100;
   1:  PR[91,1] = PR[90,1] + 49.030;
   1:  PR[91,2] = PR[90,2] + 22.972;
   1:  PR[91,3] = PR[90,3] + 93.330;
   1:L PR[91] R[100]mm/sec CNT100;
   1:  PR[91,1] = PR[90,1] + 46.902;
   1:  PR[91,2] = PR[90,2] + 24.595;
   1:  PR[91,3] = PR[90,3] + 93.341;
   1:L PR[91] R[100]mm/sec CNT100;
   1:  PR[91,1] = PR[90,1] + 42.292;
   1:  PR[91,2] = PR[90,2] + 26.928;
   1:  PR[91,3] = PR[90,3] + 93.353;
   1:L PR[91] R[100]mm/sec CNT100;
   1:  PR[91,1] = PR[90,1] + 37.245;
   1:  PR[91,2] = PR[90,2] + 28.447;
   1:  PR[91,3] = PR[90,3] + 93.376;
   1:L PR[91] R[100]mm/sec CNT100;
   1:  PR[91,1] = PR[90,1] + 32.511;
   1:  PR[91,2] = PR[90,2] + 29.043;
   1:  PR[91,3] = PR[90,3] + 93.399;
   1:L PR[91] R[100]mm/sec CNT100;
   1:  PR[91,1] = PR[90,1] + 31.765;
   1:  PR[91,2] = PR[90,2] + 29.058;
   1:  PR[91,3] = PR[90,3] + 93.421;
   1:L PR[91] R[100]mm/sec CNT100;
   1:  PR[91,1] = PR[90,1] + 27.568;
   1:  PR[91,2] = PR[90,2] + 28.827;
   1:  PR[91,3] = PR[90,3] + 93.424;
   1:L PR[91] R[100]mm/sec CNT100;
   1:  PR[91,1] = PR[90,1] + 26.159;
   1:  PR[91,2] = PR[90,2] + 28.598;
   1:  PR[91,3] = PR[90,3] + 93.443;
   1:L PR[91] R[100]mm/sec CNT100;
   1:  PR[91,1] = PR[90,1] + 21.407;
   1:  PR[91,2] = PR[90,2] + 27.464;
   1:  PR[91,3] = PR[90,3] + 93.449;
   1:L PR[91] R[100]mm/sec CNT100;
   1:  PR[91,1] = PR[90,1] + 20.575;
   1:  PR[91,2] = PR[90,2] + 27.472;
   1:  PR[91,3] = PR[90,3] + 93.471;
   1:L PR[91] R[100]mm/sec CNT100;
   1:  PR[91,1] = PR[90,1] + 19.235;
   1:  PR[91,2] = PR[90,2] + 27.410;
   1:  PR[91,3] = PR[90,3] + 93.474;
   1:L PR[91] R[100]mm/sec CNT100;
   1:  PR[91,1] = PR[90,1] + 18.275;
   1:  PR[91,2] = PR[90,2] + 27.467;
   1:  PR[91,3] = PR[90,3] + 93.480;
   1:L PR[91] R[100]mm/sec CNT100;
   1:  PR[91,1] = PR[90,1] + 7.525;
   1:  PR[91,2] = PR[90,2] + 27.884;
   1:  PR[91,3] = PR[90,3] + 93.485;
   1:L PR[91] R[100]mm/sec CNT100;
   1:  PR[91,1] = PR[90,1] + -2.993;
   1:  PR[91,2] = PR[90,2] + 27.478;
   1:  PR[91,3] = PR[90,3] + 93.533;
   1:L PR[91] R[100]mm/sec CNT100;
   1:  PR[91,1] = PR[90,1] + -5.796;
   1:  PR[91,2] = PR[90,2] + 27.186;
   1:  PR[91,3] = PR[90,3] + 93.579;
   1:L PR[91] R[100]mm/sec CNT100;
   1:  PR[91,1] = PR[90,1] + -13.027;
   1:  PR[91,2] = PR[90,2] + 26.396;
   1:  PR[91,3] = PR[90,3] + 93.592;
   1:L PR[91] R[100]mm/sec CNT100;
   1:  PR[91,1] = PR[90,1] + -18.279;
   1:  PR[91,2] = PR[90,2] + 25.461;
   1:  PR[91,3] = PR[90,3] + 93.624;
   1:L PR[91] R[100]mm/sec CNT100;
   1:  PR[91,1] = PR[90,1] + -22.384;
   1:  PR[91,2] = PR[90,2] + 24.710;
   1:  PR[91,3] = PR[90,3] + 93.648;
   1:L PR[91] R[100]mm/sec CNT100;
   1:  PR[91,1] = PR[90,1] + -30.899;
   1:  PR[91,2] = PR[90,2] + 22.489;
   1:  PR[91,3] = PR[90,3] + 93.667;
   1:L PR[91] R[100]mm/sec CNT100;
   1:  PR[91,1] = PR[90,1] + -36.804;
   1:  PR[91,2] = PR[90,2] + 20.391;
   1:  PR[91,3] = PR[90,3] + 93.706;
   1:L PR[91] R[100]mm/sec CNT100;
   1:  PR[91,1] = PR[90,1] + -37.835;
   1:  PR[91,2] = PR[90,2] + 19.997;
   1:  PR[91,3] = PR[90,3] + 93.734;
   1:L PR[91] R[100]mm/sec CNT100;
   1:  PR[91,1] = PR[90,1] + -38.951;
   1:  PR[91,2] = PR[90,2] + 19.482;
   1:  PR[91,3] = PR[90,3] + 93.739;
   1:L PR[91] R[100]mm/sec CNT100;
   1:  PR[91,1] = PR[90,1] + -43.041;
   1:  PR[91,2] = PR[90,2] + 17.397;
   1:  PR[91,3] = PR[90,3] + 93.744;
   1:L PR[91] R[100]mm/sec CNT100;
   1:  PR[91,1] = PR[90,1] + -48.727;
   1:  PR[91,2] = PR[90,2] + 13.596;
   1:  PR[91,3] = PR[90,3] + 93.765;
   1:L PR[91] R[100]mm/sec CNT100;
   1:  PR[91] = PR[90];
   1:  PR[91,1] = PR[90,1] + -49.365;
   1:  PR[91,2] = PR[90,2] + 11.172;
   1:  PR[91,3] = PR[90,3] + 95.095;
   1:L PR[91] R[100]mm/sec CNT100;
   1:  PR[91,1] = PR[90,1] + -51.153;
   1:  PR[91,2] = PR[90,2] + 9.107;
   1:  PR[91,3] = PR[90,3] + 93.811;
   1:L PR[91] R[100]mm/sec CNT100;
   1:  PR[91,1] = PR[90,1] + -51.534;
   1:  PR[91,2] = PR[90,2] + 8.367;
   1:  PR[91,3] = PR[90,3] + 93.823;
   1:L PR[91] R[100]mm/sec CNT100;
   1:  PR[91,1] = PR[90,1] + -53.546;
   1:  PR[91,2] = PR[90,2] + 4.268;
   1:  PR[91,3] = PR[90,3] + 93.827;
   1:L PR[91] R[100]mm/sec CNT100;
   1:  PR[91,1] = PR[90,1] + -53.848;
   1:  PR[91,2] = PR[90,2] + 2.477;
   1:  PR[91,3] = PR[90,3] + 93.847;
   1:L PR[91] R[100]mm/sec CNT100;
   1:  PR[91,1] = PR[90,1] + -54.520;
   1:  PR[91,2] = PR[90,2] + -0.745;
   1:  PR[91,3] = PR[90,3] + 93.856;
   1:L PR[91] R[100]mm/sec CNT100;
   1:  PR[91,1] = PR[90,1] + -54.513;
   1:  PR[91,2] = PR[90,2] + -0.783;
   1:  PR[91,3] = PR[90,3] + 93.870;
   1:L PR[91] R[100]mm/sec CNT100;
   1:  PR[91,1] = PR[90,1] + -54.240;
   1:  PR[91,2] = PR[90,2] + -1.528;
   1:  PR[91,3] = PR[90,3] + 93.871;
   1:L PR[91] R[100]mm/sec CNT100;
   1:  PR[91,1] = PR[90,1] + -53.592;
   1:  PR[91,2] = PR[90,2] + -5.660;
   1:  PR[91,3] = PR[90,3] + 93.874;
   1:L PR[91] R[100]mm/sec CNT100;
   1:  PR[91,1] = PR[90,1] + -53.290;
   1:  PR[91,2] = PR[90,2] + -6.306;
   1:  PR[91,3] = PR[90,3] + 93.893;
   1:L PR[91] R[100]mm/sec CNT100;
   1:  PR[91,1] = PR[90,1] + -51.237;
   1:  PR[91,2] = PR[90,2] + -10.564;
   1:  PR[91,3] = PR[90,3] + 93.896;
   1:L PR[91] R[100]mm/sec CNT100;
   1:  PR[91,1] = PR[90,1] + -50.866;
   1:  PR[91,2] = PR[90,2] + -11.004;
   1:  PR[91,3] = PR[90,3] + 93.917;
   1:L PR[91] R[100]mm/sec CNT100;
   1:  PR[91,1] = PR[90,1] + -47.495;
   1:  PR[91,2] = PR[90,2] + -14.421;
   1:  PR[91,3] = PR[90,3] + 93.920;
   1:L PR[91] R[100]mm/sec CNT100;
   1:  PR[91,1] = PR[90,1] + -46.719;
   1:  PR[91,2] = PR[90,2] + -15.165;
   1:  PR[91,3] = PR[90,3] + 93.942;
   1:L PR[91] R[100]mm/sec CNT100;
   1:  PR[91,1] = PR[90,1] + -44.576;
   1:  PR[91,2] = PR[90,2] + -16.660;
   1:  PR[91,3] = PR[90,3] + 93.946;
   1:L PR[91] R[100]mm/sec CNT100;
   1:  PR[91,1] = PR[90,1] + -41.398;
   1:  PR[91,2] = PR[90,2] + -18.787;
   1:  PR[91,3] = PR[90,3] + 93.958;
   1:L PR[91] R[100]mm/sec CNT100;
   1:  PR[91,1] = PR[90,1] + -37.258;
   1:  PR[91,2] = PR[90,2] + -20.921;
   1:  PR[91,3] = PR[90,3] + 93.975;
   1:L PR[91] R[100]mm/sec CNT100;
   1:  PR[91,1] = PR[90,1] + -36.150;
   1:  PR[91,2] = PR[90,2] + -21.445;
   1:  PR[91,3] = PR[90,3] + 93.996;
   1:L PR[91] R[100]mm/sec CNT100;
   1:  PR[91,1] = PR[90,1] + -28.560;
   1:  PR[91,2] = PR[90,2] + -24.144;
   1:  PR[91,3] = PR[90,3] + 94.002;
   1:L PR[91] R[100]mm/sec CNT100;
   1:  PR[91,1] = PR[90,1] + -19.983;
   1:  PR[91,2] = PR[90,2] + -26.385;
   1:  PR[91,3] = PR[90,3] + 94.038;
   1:L PR[91] R[100]mm/sec CNT100;
   1:  PR[91,1] = PR[90,1] + -15.009;
   1:  PR[91,2] = PR[90,2] + -27.294;
   1:  PR[91,3] = PR[90,3] + 94.078;
   1:L PR[91] R[100]mm/sec CNT100;
   1:  PR[91,1] = PR[90,1] + -10.557;
   1:  PR[91,2] = PR[90,2] + -28.087;
   1:  PR[91,3] = PR[90,3] + 94.101;
   1:L PR[91] R[100]mm/sec CNT100;
   1:  PR[91,1] = PR[90,1] + -0.444;
   1:  PR[91,2] = PR[90,2] + -29.181;
   1:  PR[91,3] = PR[90,3] + 94.121;
   1:L PR[91] R[100]mm/sec CNT100;
   1:  PR[91,1] = PR[90,1] + 6.896;
   1:  PR[91,2] = PR[90,2] + -29.464;
   1:  PR[91,3] = PR[90,3] + 94.167;
   1:L PR[91] R[100]mm/sec CNT100;
   1:  PR[91,1] = PR[90,1] + 9.665;
   1:  PR[91,2] = PR[90,2] + -29.600;
   1:  PR[91,3] = PR[90,3] + 94.200;
   1:L PR[91] R[100]mm/sec CNT100;
   1:  PR[91,1] = PR[90,1] + 13.880;
   1:  PR[91,2] = PR[90,2] + -29.451;
   1:  PR[91,3] = PR[90,3] + 94.212;
   1:L PR[91] R[100]mm/sec CNT100;
   1:  PR[91,1] = PR[90,1] + 21.353;
   1:  PR[91,2] = PR[90,2] + -29.130;
   1:  PR[91,3] = PR[90,3] + 94.231;
   1:L PR[91] R[100]mm/sec CNT100;
   1:  PR[91,1] = PR[90,1] + 25.563;
   1:  PR[91,2] = PR[90,2] + -30.127;
   1:  PR[91,3] = PR[90,3] + 94.265;
   1:L PR[91] R[100]mm/sec CNT100;
   1:  PR[91,1] = PR[90,1] + 27.869;
   1:  PR[91,2] = PR[90,2] + -30.501;
   1:  PR[91,3] = PR[90,3] + 94.284;
   1:L PR[91] R[100]mm/sec CNT100;
   1:  PR[91,1] = PR[90,1] + 31.160;
   1:  PR[91,2] = PR[90,2] + -30.682;
   1:  PR[91,3] = PR[90,3] + 94.295;
   1:L PR[91] R[100]mm/sec CNT100;
   1:  PR[91,1] = PR[90,1] + 32.947;
   1:  PR[91,2] = PR[90,2] + -30.648;
   1:  PR[91,3] = PR[90,3] + 94.310;
   1:L PR[91] R[100]mm/sec CNT100;
   1:  PR[91,1] = PR[90,1] + 36.769;
   1:  PR[91,2] = PR[90,2] + -30.166;
   1:  PR[91,3] = PR[90,3] + 94.318;
   1:L PR[91] R[100]mm/sec CNT100;
   1:  PR[91,1] = PR[90,1] + 37.799;
   1:  PR[91,2] = PR[90,2] + -29.954;
   1:  PR[91,3] = PR[90,3] + 94.335;
   1:L PR[91] R[100]mm/sec CNT100;
   1:  PR[91,1] = PR[90,1] + 42.128;
   1:  PR[91,2] = PR[90,2] + -28.597;
   1:  PR[91,3] = PR[90,3] + 94.340;
   1:L PR[91] R[100]mm/sec CNT100;
   1:  PR[91,1] = PR[90,1] + 42.265;
   1:  PR[91,2] = PR[90,2] + -28.541;
   1:  PR[91,3] = PR[90,3] + 94.360;
   1:L PR[91] R[100]mm/sec CNT100;
   1:  PR[91,1] = PR[90,1] + 43.627;
   1:  PR[91,2] = PR[90,2] + -27.829;
   1:  PR[91,3] = PR[90,3] + 94.361;
   1:L PR[91] R[100]mm/sec CNT100;
   1:  PR[91,1] = PR[90,1] + 46.813;
   1:  PR[91,2] = PR[90,2] + -26.224;
   1:  PR[91,3] = PR[90,3] + 94.368;
   1:L PR[91] R[100]mm/sec CNT100;
   1:  PR[91,1] = PR[90,1] + 50.933;
   1:  PR[91,2] = PR[90,2] + -23.145;
   1:  PR[91,3] = PR[90,3] + 94.384;
   1:L PR[91] R[100]mm/sec CNT100;
   1:  PR[91,1] = PR[90,1] + 52.529;
   1:  PR[91,2] = PR[90,2] + -21.411;
   1:  PR[91,3] = PR[90,3] + 94.407;
   1:L PR[91] R[100]mm/sec CNT100;
   1:  PR[91,1] = PR[90,1] + 54.411;
   1:  PR[91,2] = PR[90,2] + -19.423;
   1:  PR[91,3] = PR[90,3] + 94.418;
   1:L PR[91] R[100]mm/sec CNT100;
   1:  PR[91,1] = PR[90,1] + 56.574;
   1:  PR[91,2] = PR[90,2] + -16.056;
   1:  PR[91,3] = PR[90,3] + 94.430;
   1:L PR[91] R[100]mm/sec CNT100;
   1:  PR[91,1] = PR[90,1] + 57.151;
   1:  PR[91,2] = PR[90,2] + -15.186;
   1:  PR[91,3] = PR[90,3] + 94.448;
   1:L PR[91] R[100]mm/sec CNT100;
   1:  PR[91,1] = PR[90,1] + 58.813;
   1:  PR[91,2] = PR[90,2] + -11.280;
   1:  PR[91,3] = PR[90,3] + 94.453;
   1:L PR[91] R[100]mm/sec CNT100;
   1:  PR[91,1] = PR[90,1] + 59.145;
   1:  PR[91,2] = PR[90,2] + -10.551;
   1:  PR[91,3] = PR[90,3] + 94.472;
   1:L PR[91] R[100]mm/sec CNT100;
   1:  PR[91,1] = PR[90,1] + 60.403;
   1:  PR[91,2] = PR[90,2] + -5.711;
   1:  PR[91,3] = PR[90,3] + 94.475;
   1:L PR[91] R[100]mm/sec CNT100;
   1:  PR[91,1] = PR[90,1] + 60.481;
   1:  PR[91,2] = PR[90,2] + -4.788;
   1:  PR[91,3] = PR[90,3] + 94.498;
   1:L PR[91] R[100]mm/sec CNT100;
   1:  PR[91,1] = PR[90,1] + 60.550;
   1:  PR[91,2] = PR[90,2] + -3.505;
   1:  PR[91,3] = PR[90,3] + 94.502;
   1:L PR[91] R[100]mm/sec CNT100;
   1:  PR[91,1] = PR[90,1] + 60.782;
   1:  PR[91,2] = PR[90,2] + -0.697;
   1:  PR[91,3] = PR[90,3] + 94.508;
   1:L PR[91] R[100]mm/sec CNT100;
   1:  PR[91,1] = PR[90,1] + 60.735;
   1:  PR[91,2] = PR[90,2] + 0.247;
   1:  PR[91,3] = PR[90,3] + 94.521;
   1:L PR[91] R[100]mm/sec CNT100;
   1:  PR[91,1] = PR[90,1] + 60.403;
   1:  PR[91,2] = PR[90,2] + 4.253;
   1:  PR[91,3] = PR[90,3] + 94.525;
   1:L PR[91] R[100]mm/sec CNT100;
   1:  PR[91,1] = PR[90,1] + 59.145;
   1:  PR[91,2] = PR[90,2] + 9.092;
   1:  PR[91,3] = PR[90,3] + 94.543;
   1:L PR[91] R[100]mm/sec CNT100;
   1:  PR[91,1] = PR[90,1] + 58.813;
   1:  PR[91,2] = PR[90,2] + 9.821;
   1:  PR[91,3] = PR[90,3] + 94.565;
   1:L PR[91] R[100]mm/sec CNT100;
   1:  PR[91,1] = PR[90,1] + 57.151;
   1:  PR[91,2] = PR[90,2] + 13.728;
   1:  PR[91,3] = PR[90,3] + 94.569;
   1:L PR[91] R[100]mm/sec CNT100;
   1:  PR[91,1] = PR[90,1] + 56.574;
   1:  PR[91,2] = PR[90,2] + 14.597;
   1:  PR[91,3] = PR[90,3] + 94.588;
   1:L PR[91] R[100]mm/sec CNT100;
   1:  PR[91,1] = PR[90,1] + 54.411;
   1:  PR[91,2] = PR[90,2] + 17.964;
   1:  PR[91,3] = PR[90,3] + 94.593;
   1:L PR[91] R[100]mm/sec CNT100;
   1:  PR[91,1] = PR[90,1] + 52.529;
   1:  PR[91,2] = PR[90,2] + 19.953;
   1:  PR[91,3] = PR[90,3] + 94.611;
   1:L PR[91] R[100]mm/sec CNT100;
   1:  PR[91,1] = PR[90,1] + 50.933;
   1:  PR[91,2] = PR[90,2] + 21.686;
   1:  PR[91,3] = PR[90,3] + 94.623;
   1:L PR[91] R[100]mm/sec CNT100;
   1:  PR[91,1] = PR[90,1] + 46.813;
   1:  PR[91,2] = PR[90,2] + 24.766;
   1:  PR[91,3] = PR[90,3] + 94.634;
   1:L PR[91] R[100]mm/sec CNT100;
   1:  PR[91,1] = PR[90,1] + 43.627;
   1:  PR[91,2] = PR[90,2] + 26.370;
   1:  PR[91,3] = PR[90,3] + 94.657;
   1:L PR[91] R[100]mm/sec CNT100;
   1:  PR[91,1] = PR[90,1] + 42.266;
   1:  PR[91,2] = PR[90,2] + 27.082;
   1:  PR[91,3] = PR[90,3] + 94.673;
   1:L PR[91] R[100]mm/sec CNT100;
   1:  PR[91,1] = PR[90,1] + 42.128;
   1:  PR[91,2] = PR[90,2] + 27.139;
   1:  PR[91,3] = PR[90,3] + 94.680;
   1:L PR[91] R[100]mm/sec CNT100;
   1:  PR[91,1] = PR[90,1] + 37.800;
   1:  PR[91,2] = PR[90,2] + 28.494;
   1:L PR[91] R[100]mm/sec CNT100;
   1:  PR[91,1] = PR[90,1] + 36.772;
   1:  PR[91,2] = PR[90,2] + 28.707;
   1:  PR[91,3] = PR[90,3] + 94.701;
   1:L PR[91] R[100]mm/sec CNT100;
   1:  PR[91,1] = PR[90,1] + 32.950;
   1:  PR[91,2] = PR[90,2] + 29.189;
   1:  PR[91,3] = PR[90,3] + 94.706;
   1:L PR[91] R[100]mm/sec CNT100;
   1:  PR[91,1] = PR[90,1] + 31.164;
   1:  PR[91,2] = PR[90,2] + 29.224;
   1:  PR[91,3] = PR[90,3] + 94.723;
   1:L PR[91] R[100]mm/sec CNT100;
   1:  PR[91,1] = PR[90,1] + 27.875;
   1:  PR[91,2] = PR[90,2] + 29.043;
   1:  PR[91,3] = PR[90,3] + 94.731;
   1:L PR[91] R[100]mm/sec CNT100;
   1:  PR[91,1] = PR[90,1] + 25.550;
   1:  PR[91,2] = PR[90,2] + 28.666;
   1:  PR[91,3] = PR[90,3] + 94.746;
   1:L PR[91] R[100]mm/sec CNT100;
   1:  PR[91,1] = PR[90,1] + 21.358;
   1:  PR[91,2] = PR[90,2] + 27.673;
   1:  PR[91,3] = PR[90,3] + 94.756;
   1:L PR[91] R[100]mm/sec CNT100;
   1:  PR[91,1] = PR[90,1] + 9.661;
   1:  PR[91,2] = PR[90,2] + 28.141;
   1:  PR[91,3] = PR[90,3] + 94.776;
   1:L PR[91] R[100]mm/sec CNT100;
   1:  PR[91,1] = PR[90,1] + 6.896;
   1:  PR[91,2] = PR[90,2] + 28.005;
   1:  PR[91,3] = PR[90,3] + 94.828;
   1:L PR[91] R[100]mm/sec CNT100;
   1:  PR[91,1] = PR[90,1] + -0.444;
   1:  PR[91,2] = PR[90,2] + 27.723;
   1:  PR[91,3] = PR[90,3] + 94.841;
   1:L PR[91] R[100]mm/sec CNT100;
   1:  PR[91,1] = PR[90,1] + -10.557;
   1:  PR[91,2] = PR[90,2] + 26.628;
   1:  PR[91,3] = PR[90,3] + 94.874;
   1:L PR[91] R[100]mm/sec CNT100;
   1:  PR[91,1] = PR[90,1] + -15.009;
   1:  PR[91,2] = PR[90,2] + 25.835;
   1:  PR[91,3] = PR[90,3] + 94.920;
   1:L PR[91] R[100]mm/sec CNT100;
   1:  PR[91,1] = PR[90,1] + -19.983;
   1:  PR[91,2] = PR[90,2] + 24.926;
   1:  PR[91,3] = PR[90,3] + 94.940;
   1:L PR[91] R[100]mm/sec CNT100;
   1:  PR[91,1] = PR[90,1] + -28.560;
   1:  PR[91,2] = PR[90,2] + 22.685;
   1:  PR[91,3] = PR[90,3] + 94.963;
   1:L PR[91] R[100]mm/sec CNT100;
   1:  PR[91,1] = PR[90,1] + -36.150;
   1:  PR[91,2] = PR[90,2] + 19.987;
   1:  PR[91,3] = PR[90,3] + 95.003;
   1:L PR[91] R[100]mm/sec CNT100;
   1:  PR[91,1] = PR[90,1] + -37.263;
   1:  PR[91,2] = PR[90,2] + 19.461;
   1:  PR[91,3] = PR[90,3] + 95.039;
   1:L PR[91] R[100]mm/sec CNT100;
   1:  PR[91,1] = PR[90,1] + -41.425;
   1:  PR[91,2] = PR[90,2] + 17.338;
   1:  PR[91,3] = PR[90,3] + 95.044;
   1:L PR[91] R[100]mm/sec CNT100;
   1:  PR[91,1] = PR[90,1] + -45.308;
   1:  PR[91,2] = PR[90,2] + 14.742;
   1:  PR[91,3] = PR[90,3] + 95.065;
   1:L PR[91] R[100]mm/sec CNT100;
   1:  PR[91,1] = PR[90,1] + -46.871;
   1:  PR[91,2] = PR[90,2] + 13.661;
   1:  PR[91,3] = PR[90,3] + 95.086;
   1:L PR[91] R[100]mm/sec CNT100;
   1:  PR[91] = PR[90];
   1:  PR[91,1] = PR[90,1] + -49.712;
   1:  PR[91,2] = PR[90,2] + 9.014;
   1:  PR[91,3] = PR[90,3] + 96.395;
   1:L PR[91] R[100]mm/sec CNT100;
   1:  PR[91,1] = PR[90,1] + -49.895;
   1:  PR[91,2] = PR[90,2] + 8.687;
   1:  PR[91,3] = PR[90,3] + 95.126;
   1:L PR[91] R[100]mm/sec CNT100;
   1:  PR[91,1] = PR[90,1] + -52.067;
   1:  PR[91,2] = PR[90,2] + 4.259;
   1:  PR[91,3] = PR[90,3] + 95.127;
   1:L PR[91] R[100]mm/sec CNT100;
   1:  PR[91,1] = PR[90,1] + -52.198;
   1:  PR[91,2] = PR[90,2] + 3.486;
   1:  PR[91,3] = PR[90,3] + 95.150;
   1:L PR[91] R[100]mm/sec CNT100;
   1:  PR[91,1] = PR[90,1] + -52.873;
   1:  PR[91,2] = PR[90,2] + 0.250;
   1:  PR[91,3] = PR[90,3] + 95.153;
   1:L PR[91] R[100]mm/sec CNT100;
   1:  PR[91,1] = PR[90,1] + -53.010;
   1:  PR[91,2] = PR[90,2] + -0.543;
   1:  PR[91,3] = PR[90,3] + 95.168;
   1:L PR[91] R[100]mm/sec CNT100;
   1:  PR[91,1] = PR[90,1] + -52.918;
   1:  PR[91,2] = PR[90,2] + -0.793;
   1:  PR[91,3] = PR[90,3] + 95.172;
   1:L PR[91] R[100]mm/sec CNT100;
   1:  PR[91,1] = PR[90,1] + -52.146;
   1:  PR[91,2] = PR[90,2] + -5.720;
   1:  PR[91,3] = PR[90,3] + 95.173;
   1:L PR[91] R[100]mm/sec CNT100;
   1:  PR[91,1] = PR[90,1] + -51.429;
   1:  PR[91,2] = PR[90,2] + -7.208;
   1:  PR[91,3] = PR[90,3] + 95.196;
   1:L PR[91] R[100]mm/sec CNT100;
   1:  PR[91,1] = PR[90,1] + -49.680;
   1:  PR[91,2] = PR[90,2] + -10.338;
   1:  PR[91,3] = PR[90,3] + 95.203;
   1:L PR[91] R[100]mm/sec CNT100;
   1:  PR[91,1] = PR[90,1] + -49.463;
   1:  PR[91,2] = PR[90,2] + -10.639;
   1:  PR[91,3] = PR[90,3] + 95.219;
   1:L PR[91] R[100]mm/sec CNT100;
   1:  PR[91,1] = PR[90,1] + -46.177;
   1:  PR[91,2] = PR[90,2] + -13.970;
   1:  PR[91,3] = PR[90,3] + 95.221;
   1:L PR[91] R[100]mm/sec CNT100;
   1:  PR[91,1] = PR[90,1] + -44.827;
   1:  PR[91,2] = PR[90,2] + -15.265;
   1:  PR[91,3] = PR[90,3] + 95.242;
   1:L PR[91] R[100]mm/sec CNT100;
   1:  PR[91,1] = PR[90,1] + -41.238;
   1:  PR[91,2] = PR[90,2] + -17.768;
   1:  PR[91,3] = PR[90,3] + 95.251;
   1:L PR[91] R[100]mm/sec CNT100;
   1:  PR[91,1] = PR[90,1] + -39.794;
   1:  PR[91,2] = PR[90,2] + -18.734;
   1:  PR[91,3] = PR[90,3] + 95.270;
   1:L PR[91] R[100]mm/sec CNT100;
   1:  PR[91,1] = PR[90,1] + -37.907;
   1:  PR[91,2] = PR[90,2] + -19.708;
   1:  PR[91,3] = PR[90,3] + 95.278;
   1:L PR[91] R[100]mm/sec CNT100;
   1:  PR[91,1] = PR[90,1] + -33.865;
   1:  PR[91,2] = PR[90,2] + -21.618;
   1:  PR[91,3] = PR[90,3] + 95.288;
   1:L PR[91] R[100]mm/sec CNT100;
   1:  PR[91,1] = PR[90,1] + -26.220;
   1:  PR[91,2] = PR[90,2] + -24.340;
   1:  PR[91,3] = PR[90,3] + 95.308;
   1:L PR[91] R[100]mm/sec CNT100;
   1:  PR[91,1] = PR[90,1] + -17.581;
   1:  PR[91,2] = PR[90,2] + -26.600;
   1:  PR[91,3] = PR[90,3] + 95.345;
   1:L PR[91] R[100]mm/sec CNT100;
   1:  PR[91,1] = PR[90,1] + -11.739;
   1:  PR[91,2] = PR[90,2] + -27.669;
   1:  PR[91,3] = PR[90,3] + 95.385;
   1:L PR[91] R[100]mm/sec CNT100;
   1:  PR[91,1] = PR[90,1] + -8.086;
   1:  PR[91,2] = PR[90,2] + -28.319;
   1:  PR[91,3] = PR[90,3] + 95.412;
   1:L PR[91] R[100]mm/sec CNT100;
   1:  PR[91,1] = PR[90,1] + 1.029;
   1:  PR[91,2] = PR[90,2] + -29.314;
   1:  PR[91,3] = PR[90,3] + 95.429;
   1:L PR[91] R[100]mm/sec CNT100;
   1:  PR[91,1] = PR[90,1] + 2.098;
   1:  PR[91,2] = PR[90,2] + -29.426;
   1:  PR[91,3] = PR[90,3] + 95.471;
   1:L PR[91] R[100]mm/sec CNT100;
   1:  PR[91,1] = PR[90,1] + 6.247;
   1:  PR[91,2] = PR[90,2] + -29.586;
   1:  PR[91,3] = PR[90,3] + 95.475;
   1:L PR[91] R[100]mm/sec CNT100;
   1:  PR[91,1] = PR[90,1] + 11.792;
   1:  PR[91,2] = PR[90,2] + -29.857;
   1:  PR[91,3] = PR[90,3] + 95.494;
   1:L PR[91] R[100]mm/sec CNT100;
   1:  PR[91,1] = PR[90,1] + 14.899;
   1:  PR[91,2] = PR[90,2] + -29.747;
   1:  PR[91,3] = PR[90,3] + 95.519;
   1:L PR[91] R[100]mm/sec CNT100;
   1:  PR[91,1] = PR[90,1] + 20.303;
   1:  PR[91,2] = PR[90,2] + -29.520;
   1:  PR[91,3] = PR[90,3] + 95.533;
   1:L PR[91] R[100]mm/sec CNT100;
   1:  PR[91,1] = PR[90,1] + 24.444;
   1:  PR[91,2] = PR[90,2] + -29.300;
   1:  PR[91,3] = PR[90,3] + 95.558;
   1:L PR[91] R[100]mm/sec CNT100;
   1:  PR[91,1] = PR[90,1] + 24.240;
   1:  PR[91,2] = PR[90,2] + -30.026;
   1:  PR[91,3] = PR[90,3] + 95.577;
   1:L PR[91] R[100]mm/sec CNT100;
   1:  PR[91,1] = PR[90,1] + 24.959;
   1:  PR[91,2] = PR[90,2] + -30.195;
   1:  PR[91,3] = PR[90,3] + 95.580;
   1:L PR[91] R[100]mm/sec CNT100;
   1:  PR[91,1] = PR[90,1] + 28.174;
   1:  PR[91,2] = PR[90,2] + -30.717;
   1:  PR[91,3] = PR[90,3] + 95.583;
   1:L PR[91] R[100]mm/sec CNT100;
   1:  PR[91,1] = PR[90,1] + 30.556;
   1:  PR[91,2] = PR[90,2] + -30.848;
   1:  PR[91,3] = PR[90,3] + 95.598;
   1:L PR[91] R[100]mm/sec CNT100;
   1:  PR[91,1] = PR[90,1] + 33.384;
   1:  PR[91,2] = PR[90,2] + -30.793;
   1:  PR[91,3] = PR[90,3] + 95.609;
   1:L PR[91] R[100]mm/sec CNT100;
   1:  PR[91,1] = PR[90,1] + 36.206;
   1:  PR[91,2] = PR[90,2] + -30.438;
   1:  PR[91,3] = PR[90,3] + 95.622;
   1:L PR[91] R[100]mm/sec CNT100;
   1:  PR[91,1] = PR[90,1] + 38.380;
   1:  PR[91,2] = PR[90,2] + -29.988;
   1:  PR[91,3] = PR[90,3] + 95.635;
   1:L PR[91] R[100]mm/sec CNT100;
   1:  PR[91,1] = PR[90,1] + 41.632;
   1:  PR[91,2] = PR[90,2] + -28.969;
   1:  PR[91,3] = PR[90,3] + 95.645;
   1:L PR[91] R[100]mm/sec CNT100;
   1:  PR[91,1] = PR[90,1] + 42.997;
   1:  PR[91,2] = PR[90,2] + -28.411;
   1:  PR[91,3] = PR[90,3] + 95.660;
   1:L PR[91] R[100]mm/sec CNT100;
   1:  PR[91,1] = PR[90,1] + 46.615;
   1:  PR[91,2] = PR[90,2] + -26.519;
   1:  PR[91,3] = PR[90,3] + 95.667;
   1:L PR[91] R[100]mm/sec CNT100;
   1:  PR[91,1] = PR[90,1] + 47.102;
   1:  PR[91,2] = PR[90,2] + -26.205;
   1:  PR[91,3] = PR[90,3] + 95.685;
   1:L PR[91] R[100]mm/sec CNT100;
   1:  PR[91,1] = PR[90,1] + 49.866;
   1:  PR[91,2] = PR[90,2] + -24.067;
   1:  PR[91,3] = PR[90,3] + 95.688;
   1:L PR[91] R[100]mm/sec CNT100;
   1:  PR[91,1] = PR[90,1] + 50.896;
   1:  PR[91,2] = PR[90,2] + -23.301;
   1:  PR[91,3] = PR[90,3] + 95.704;
   1:L PR[91] R[100]mm/sec CNT100;
   1:  PR[91,1] = PR[90,1] + 54.418;
   1:  PR[91,2] = PR[90,2] + -19.573;
   1:  PR[91,3] = PR[90,3] + 95.710;
   1:L PR[91] R[100]mm/sec CNT100;
   1:  PR[91,1] = PR[90,1] + 55.294;
   1:  PR[91,2] = PR[90,2] + -18.209;
   1:  PR[91,3] = PR[90,3] + 95.733;
   1:L PR[91] R[100]mm/sec CNT100;
   1:  PR[91,1] = PR[90,1] + 57.216;
   1:  PR[91,2] = PR[90,2] + -15.312;
   1:  PR[91,3] = PR[90,3] + 95.740;
   1:L PR[91] R[100]mm/sec CNT100;
   1:  PR[91,1] = PR[90,1] + 58.360;
   1:  PR[91,2] = PR[90,2] + -12.623;
   1:  PR[91,3] = PR[90,3] + 95.756;
   1:L PR[91] R[100]mm/sec CNT100;
   1:  PR[91,1] = PR[90,1] + 59.226;
   1:  PR[91,2] = PR[90,2] + -10.662;
   1:  PR[91,3] = PR[90,3] + 95.769;
   1:L PR[91] R[100]mm/sec CNT100;
   1:  PR[91,1] = PR[90,1] + 60.131;
   1:  PR[91,2] = PR[90,2] + -6.926;
   1:  PR[91,3] = PR[90,3] + 95.779;
   1:L PR[91] R[100]mm/sec CNT100;
   1:  PR[91,1] = PR[90,1] + 60.428;
   1:  PR[91,2] = PR[90,2] + -5.751;
   1:  PR[91,3] = PR[90,3] + 95.796;
   1:L PR[91] R[100]mm/sec CNT100;
   1:  PR[91,1] = PR[90,1] + 60.838;
   1:  PR[91,2] = PR[90,2] + -0.729;
   1:  PR[91,3] = PR[90,3] + 95.802;
   1:L PR[91] R[100]mm/sec CNT100;
   1:  PR[91,1] = PR[90,1] + 60.428;
   1:  PR[91,2] = PR[90,2] + 4.292;
   1:  PR[91,3] = PR[90,3] + 95.825;
   1:L PR[91] R[100]mm/sec CNT100;
   1:  PR[91,1] = PR[90,1] + 60.131;
   1:  PR[91,2] = PR[90,2] + 5.467;
   1:  PR[91,3] = PR[90,3] + 95.847;
   1:L PR[91] R[100]mm/sec CNT100;
   1:  PR[91,1] = PR[90,1] + 59.226;
   1:  PR[91,2] = PR[90,2] + 9.203;
   1:  PR[91,3] = PR[90,3] + 95.853;
   1:L PR[91] R[100]mm/sec CNT100;
   1:  PR[91,1] = PR[90,1] + 58.360;
   1:  PR[91,2] = PR[90,2] + 11.164;
   1:  PR[91,3] = PR[90,3] + 95.870;
   1:L PR[91] R[100]mm/sec CNT100;
   1:  PR[91,1] = PR[90,1] + 57.216;
   1:  PR[91,2] = PR[90,2] + 13.853;
   1:  PR[91,3] = PR[90,3] + 95.880;
   1:L PR[91] R[100]mm/sec CNT100;
   1:  PR[91,1] = PR[90,1] + 55.294;
   1:  PR[91,2] = PR[90,2] + 16.750;
   1:  PR[91,3] = PR[90,3] + 95.893;
   1:L PR[91] R[100]mm/sec CNT100;
   1:  PR[91,1] = PR[90,1] + 54.418;
   1:  PR[91,2] = PR[90,2] + 18.114;
   1:  PR[91,3] = PR[90,3] + 95.909;
   1:L PR[91] R[100]mm/sec CNT100;
   1:  PR[91,1] = PR[90,1] + 50.896;
   1:  PR[91,2] = PR[90,2] + 21.842;
   1:  PR[91,3] = PR[90,3] + 95.916;
   1:L PR[91] R[100]mm/sec CNT100;
   1:  PR[91,1] = PR[90,1] + 49.866;
   1:  PR[91,2] = PR[90,2] + 22.609;
   1:  PR[91,3] = PR[90,3] + 95.940;
   1:L PR[91] R[100]mm/sec CNT100;
   1:  PR[91,1] = PR[90,1] + 47.103;
   1:  PR[91,2] = PR[90,2] + 24.746;
   1:  PR[91,3] = PR[90,3] + 95.945;
   1:L PR[91] R[100]mm/sec CNT100;
   1:  PR[91,1] = PR[90,1] + 46.616;
   1:  PR[91,2] = PR[90,2] + 25.060;
   1:  PR[91,3] = PR[90,3] + 95.961;
   1:L PR[91] R[100]mm/sec CNT100;
   1:  PR[91,1] = PR[90,1] + 42.999;
   1:  PR[91,2] = PR[90,2] + 26.952;
   1:  PR[91,3] = PR[90,3] + 95.964;
   1:L PR[91] R[100]mm/sec CNT100;
   1:  PR[91,1] = PR[90,1] + 41.635;
   1:  PR[91,2] = PR[90,2] + 27.510;
   1:  PR[91,3] = PR[90,3] + 95.982;
   1:L PR[91] R[100]mm/sec CNT100;
   1:  PR[91,1] = PR[90,1] + 38.383;
   1:  PR[91,2] = PR[90,2] + 28.528;
   1:  PR[91,3] = PR[90,3] + 95.989;
   1:L PR[91] R[100]mm/sec CNT100;
   1:  PR[91,1] = PR[90,1] + 36.211;
   1:  PR[91,2] = PR[90,2] + 28.979;
   1:  PR[91,3] = PR[90,3] + 96.004;
   1:L PR[91] R[100]mm/sec CNT100;
   1:  PR[91,1] = PR[90,1] + 33.389;
   1:  PR[91,2] = PR[90,2] + 29.334;
   1:  PR[91,3] = PR[90,3] + 96.014;
   1:L PR[91] R[100]mm/sec CNT100;
   1:  PR[91,1] = PR[90,1] + 30.562;
   1:  PR[91,2] = PR[90,2] + 29.390;
   1:  PR[91,3] = PR[90,3] + 96.027;
   1:L PR[91] R[100]mm/sec CNT100;
   1:  PR[91,1] = PR[90,1] + 28.182;
   1:  PR[91,2] = PR[90,2] + 29.258;
   1:  PR[91,3] = PR[90,3] + 96.040;
   1:L PR[91] R[100]mm/sec CNT100;
   1:  PR[91,1] = PR[90,1] + 24.943;
   1:  PR[91,2] = PR[90,2] + 28.733;
   1:  PR[91,3] = PR[90,3] + 96.051;
   1:L PR[91] R[100]mm/sec CNT100;
   1:  PR[91,1] = PR[90,1] + 21.966;
   1:  PR[91,2] = PR[90,2] + 28.031;
   1:  PR[91,3] = PR[90,3] + 96.066;
   1:L PR[91] R[100]mm/sec CNT100;
   1:  PR[91,1] = PR[90,1] + 20.333;
   1:  PR[91,2] = PR[90,2] + 28.060;
   1:  PR[91,3] = PR[90,3] + 96.080;
   1:L PR[91] R[100]mm/sec CNT100;
   1:  PR[91,1] = PR[90,1] + 11.788;
   1:  PR[91,2] = PR[90,2] + 28.398;
   1:  PR[91,3] = PR[90,3] + 96.087;
   1:L PR[91] R[100]mm/sec CNT100;
   1:  PR[91,1] = PR[90,1] + 6.247;
   1:  PR[91,2] = PR[90,2] + 28.127;
   1:  PR[91,3] = PR[90,3] + 96.126;
   1:L PR[91] R[100]mm/sec CNT100;
   1:  PR[91,1] = PR[90,1] + 2.103;
   1:  PR[91,2] = PR[90,2] + 27.967;
   1:  PR[91,3] = PR[90,3] + 96.151;
   1:L PR[91] R[100]mm/sec CNT100;
   1:  PR[91,1] = PR[90,1] + -8.086;
   1:  PR[91,2] = PR[90,2] + 26.860;
   1:  PR[91,3] = PR[90,3] + 96.170;
   1:L PR[91] R[100]mm/sec CNT100;
   1:  PR[91,1] = PR[90,1] + -11.739;
   1:  PR[91,2] = PR[90,2] + 26.210;
   1:  PR[91,3] = PR[90,3] + 96.216;
   1:L PR[91] R[100]mm/sec CNT100;
   1:  PR[91,1] = PR[90,1] + -17.583;
   1:  PR[91,2] = PR[90,2] + 25.141;
   1:  PR[91,3] = PR[90,3] + 96.233;
   1:L PR[91] R[100]mm/sec CNT100;
   1:  PR[91,1] = PR[90,1] + -23.182;
   1:  PR[91,2] = PR[90,2] + 23.686;
   1:  PR[91,3] = PR[90,3] + 96.260;
   1:L PR[91] R[100]mm/sec CNT100;
   1:  PR[91,1] = PR[90,1] + -26.217;
   1:  PR[91,2] = PR[90,2] + 22.882;
   1:  PR[91,3] = PR[90,3] + 96.286;
   1:L PR[91] R[100]mm/sec CNT100;
   1:  PR[91,1] = PR[90,1] + -33.865;
   1:  PR[91,2] = PR[90,2] + 20.160;
   1:  PR[91,3] = PR[90,3] + 96.300;
   1:L PR[91] R[100]mm/sec CNT100;
   1:  PR[91,1] = PR[90,1] + -37.911;
   1:  PR[91,2] = PR[90,2] + 18.247;
   1:  PR[91,3] = PR[90,3] + 96.337;
   1:L PR[91] R[100]mm/sec CNT100;
   1:  PR[91,1] = PR[90,1] + -39.809;
   1:  PR[91,2] = PR[90,2] + 17.279;
   1:  PR[91,3] = PR[90,3] + 96.357;
   1:L PR[91] R[100]mm/sec CNT100;
   1:  PR[91,1] = PR[90,1] + -41.586;
   1:  PR[91,2] = PR[90,2] + 16.091;
   1:  PR[91,3] = PR[90,3] + 96.367;
   1:L PR[91] R[100]mm/sec CNT100;
   1:  PR[91,1] = PR[90,1] + -44.936;
   1:  PR[91,2] = PR[90,2] + 13.774;
   1:  PR[91,3] = PR[90,3] + 96.377;
   1:L PR[91] R[100]mm/sec CNT100;
   1:  PR[91] = PR[90];
   1:  PR[91,1] = PR[90,1] + -46.060;
   1:  PR[91,2] = PR[90,2] + 10.834;
   1:  PR[91,3] = PR[90,3] + 97.695;
   1:L PR[91] R[100]mm/sec CNT100;
   1:  PR[91,1] = PR[90,1] + -47.622;
   1:  PR[91,2] = PR[90,2] + 9.323;
   1:  PR[91,3] = PR[90,3] + 96.415;
   1:L PR[91] R[100]mm/sec CNT100;
   1:  PR[91,1] = PR[90,1] + -48.087;
   1:  PR[91,2] = PR[90,2] + 8.684;
   1:  PR[91,3] = PR[90,3] + 96.425;
   1:L PR[91] R[100]mm/sec CNT100;
   1:  PR[91,1] = PR[90,1] + -50.599;
   1:  PR[91,2] = PR[90,2] + 4.195;
   1:  PR[91,3] = PR[90,3] + 96.428;
   1:L PR[91] R[100]mm/sec CNT100;
   1:  PR[91,1] = PR[90,1] + -51.439;
   1:  PR[91,2] = PR[90,2] + -0.728;
   1:  PR[91,3] = PR[90,3] + 96.452;
   1:L PR[91] R[100]mm/sec CNT100;
   1:  PR[91,1] = PR[90,1] + -51.125;
   1:  PR[91,2] = PR[90,2] + -2.557;
   1:  PR[91,3] = PR[90,3] + 96.475;
   1:L PR[91] R[100]mm/sec CNT100;
   1:  PR[91,1] = PR[90,1] + -50.510;
   1:  PR[91,2] = PR[90,2] + -5.430;
   1:  PR[91,3] = PR[90,3] + 96.483;
   1:L PR[91] R[100]mm/sec CNT100;
   1:  PR[91,1] = PR[90,1] + -50.477;
   1:  PR[91,2] = PR[90,2] + -5.674;
   1:  PR[91,3] = PR[90,3] + 96.497;
   1:L PR[91] R[100]mm/sec CNT100;
   1:  PR[91,1] = PR[90,1] + -50.419;
   1:  PR[91,2] = PR[90,2] + -5.812;
   1:  PR[91,3] = PR[90,3] + 96.498;
   1:L PR[91] R[100]mm/sec CNT100;
   1:  PR[91,1] = PR[90,1] + -48.096;
   1:  PR[91,2] = PR[90,2] + -9.970;
   1:L PR[91] R[100]mm/sec CNT100;
   1:  PR[91,1] = PR[90,1] + -47.381;
   1:  PR[91,2] = PR[90,2] + -10.962;
   1:  PR[91,3] = PR[90,3] + 96.520;
   1:L PR[91] R[100]mm/sec CNT100;
   1:  PR[91,1] = PR[90,1] + -44.859;
   1:  PR[91,2] = PR[90,2] + -13.519;
   1:  PR[91,3] = PR[90,3] + 96.526;
   1:L PR[91] R[100]mm/sec CNT100;
   1:  PR[91,1] = PR[90,1] + -42.934;
   1:  PR[91,2] = PR[90,2] + -15.364;
   1:  PR[91,3] = PR[90,3] + 96.542;
   1:L PR[91] R[100]mm/sec CNT100;
   1:  PR[91,1] = PR[90,1] + -38.335;
   1:  PR[91,2] = PR[90,2] + -18.573;
   1:  PR[91,3] = PR[90,3] + 96.554;
   1:L PR[91] R[100]mm/sec CNT100;
   1:  PR[91,1] = PR[90,1] + -38.178;
   1:  PR[91,2] = PR[90,2] + -18.672;
   1:  PR[91,3] = PR[90,3] + 96.580;
   1:L PR[91] R[100]mm/sec CNT100;
   1:  PR[91,1] = PR[90,1] + -31.581;
   1:  PR[91,2] = PR[90,2] + -21.791;
   1:  PR[91,3] = PR[90,3] + 96.581;
   1:L PR[91] R[100]mm/sec CNT100;
   1:  PR[91,1] = PR[90,1] + -23.878;
   1:  PR[91,2] = PR[90,2] + -24.537;
   1:  PR[91,3] = PR[90,3] + 96.614;
   1:L PR[91] R[100]mm/sec CNT100;
   1:  PR[91,1] = PR[90,1] + -20.066;
   1:  PR[91,2] = PR[90,2] + -25.546;
   1:  PR[91,3] = PR[90,3] + 96.652;
   1:L PR[91] R[100]mm/sec CNT100;
   1:  PR[91,1] = PR[90,1] + -15.183;
   1:  PR[91,2] = PR[90,2] + -26.815;
   1:  PR[91,3] = PR[90,3] + 96.670;
   1:L PR[91] R[100]mm/sec CNT100;
   1:  PR[91,1] = PR[90,1] + -5.612;
   1:  PR[91,2] = PR[90,2] + -28.552;
   1:  PR[91,3] = PR[90,3] + 96.693;
   1:L PR[91] R[100]mm/sec CNT100;
   1:  PR[91,1] = PR[90,1] + 4.658;
   1:  PR[91,2] = PR[90,2] + -29.672;
   1:  PR[91,3] = PR[90,3] + 96.737;
   1:L PR[91] R[100]mm/sec CNT100;
   1:  PR[91,1] = PR[90,1] + 13.913;
   1:  PR[91,2] = PR[90,2] + -30.115;
   1:  PR[91,3] = PR[90,3] + 96.785;
   1:L PR[91] R[100]mm/sec CNT100;
   1:  PR[91,1] = PR[90,1] + 19.447;
   1:  PR[91,2] = PR[90,2] + -29.895;
   1:  PR[91,3] = PR[90,3] + 96.827;
   1:L PR[91] R[100]mm/sec CNT100;
   1:  PR[91,1] = PR[90,1] + 25.046;
   1:  PR[91,2] = PR[90,2] + -29.598;
   1:  PR[91,3] = PR[90,3] + 96.852;
   1:L PR[91] R[100]mm/sec CNT100;
   1:  PR[91,1] = PR[90,1] + 24.837;
   1:  PR[91,2] = PR[90,2] + -30.342;
   1:  PR[91,3] = PR[90,3] + 96.878;
   1:L PR[91] R[100]mm/sec CNT100;
   1:  PR[91,1] = PR[90,1] + 28.479;
   1:  PR[91,2] = PR[90,2] + -30.933;
   1:  PR[91,3] = PR[90,3] + 96.881;
   1:L PR[91] R[100]mm/sec CNT100;
   1:  PR[91,1] = PR[90,1] + 29.952;
   1:  PR[91,2] = PR[90,2] + -31.014;
   1:  PR[91,3] = PR[90,3] + 96.898;
   1:L PR[91] R[100]mm/sec CNT100;
   1:  PR[91,1] = PR[90,1] + 33.821;
   1:  PR[91,2] = PR[90,2] + -30.939;
   1:  PR[91,3] = PR[90,3] + 96.905;
   1:L PR[91] R[100]mm/sec CNT100;
   1:  PR[91,1] = PR[90,1] + 35.643;
   1:  PR[91,2] = PR[90,2] + -30.709;
   1:  PR[91,3] = PR[90,3] + 96.923;
   1:L PR[91] R[100]mm/sec CNT100;
   1:  PR[91,1] = PR[90,1] + 38.961;
   1:  PR[91,2] = PR[90,2] + -30.023;
   1:  PR[91,3] = PR[90,3] + 96.931;
   1:L PR[91] R[100]mm/sec CNT100;
   1:  PR[91,1] = PR[90,1] + 41.137;
   1:  PR[91,2] = PR[90,2] + -29.341;
   1:  PR[91,3] = PR[90,3] + 96.947;
   1:L PR[91] R[100]mm/sec CNT100;
   1:  PR[91,1] = PR[90,1] + 43.729;
   1:  PR[91,2] = PR[90,2] + -28.282;
   1:  PR[91,3] = PR[90,3] + 96.957;
   1:L PR[91] R[100]mm/sec CNT100;
   1:  PR[91,1] = PR[90,1] + 46.218;
   1:  PR[91,2] = PR[90,2] + -26.980;
   1:  PR[91,3] = PR[90,3] + 96.970;
   1:L PR[91] R[100]mm/sec CNT100;
   1:  PR[91,1] = PR[90,1] + 47.983;
   1:  PR[91,2] = PR[90,2] + -25.844;
   1:  PR[91,3] = PR[90,3] + 96.983;
   1:L PR[91] R[100]mm/sec CNT100;
   1:  PR[91,1] = PR[90,1] + 50.702;
   1:  PR[91,2] = PR[90,2] + -23.741;
   1:  PR[91,3] = PR[90,3] + 96.992;
   1:L PR[91] R[100]mm/sec CNT100;
   1:  PR[91,1] = PR[90,1] + 51.627;
   1:  PR[91,2] = PR[90,2] + -22.872;
   1:  PR[91,3] = PR[90,3] + 97.008;
   1:L PR[91] R[100]mm/sec CNT100;
   1:  PR[91,1] = PR[90,1] + 54.429;
   1:  PR[91,2] = PR[90,2] + -19.791;
   1:  PR[91,3] = PR[90,3] + 97.014;
   1:L PR[91] R[100]mm/sec CNT100;
   1:  PR[91,1] = PR[90,1] + 54.623;
   1:  PR[91,2] = PR[90,2] + -19.527;
   1:  PR[91,3] = PR[90,3] + 97.033;
   1:L PR[91] R[100]mm/sec CNT100;
   1:  PR[91,1] = PR[90,1] + 55.950;
   1:  PR[91,2] = PR[90,2] + -17.444;
   1:  PR[91,3] = PR[90,3] + 97.034;
   1:L PR[91] R[100]mm/sec CNT100;
   1:  PR[91,1] = PR[90,1] + 57.287;
   1:  PR[91,2] = PR[90,2] + -15.427;
   1:  PR[91,3] = PR[90,3] + 97.046;
   1:L PR[91] R[100]mm/sec CNT100;
   1:  PR[91,1] = PR[90,1] + 59.343;
   1:  PR[91,2] = PR[90,2] + -10.755;
   1:  PR[91,3] = PR[90,3] + 97.057;
   1:L PR[91] R[100]mm/sec CNT100;
   1:  PR[91,1] = PR[90,1] + 59.644;
   1:  PR[91,2] = PR[90,2] + -9.515;
   1:  PR[91,3] = PR[90,3] + 97.080;
   1:L PR[91] R[100]mm/sec CNT100;
   1:  PR[91,1] = PR[90,1] + 60.584;
   1:  PR[91,2] = PR[90,2] + -5.800;
   1:  PR[91,3] = PR[90,3] + 97.086;
   1:L PR[91] R[100]mm/sec CNT100;
   1:  PR[91,1] = PR[90,1] + 61.001;
   1:  PR[91,2] = PR[90,2] + -0.729;
   1:  PR[91,3] = PR[90,3] + 97.103;
   1:L PR[91] R[100]mm/sec CNT100;
   1:  PR[91,1] = PR[90,1] + 60.584;
   1:  PR[91,2] = PR[90,2] + 4.341;
   1:  PR[91,3] = PR[90,3] + 97.127;
   1:L PR[91] R[100]mm/sec CNT100;
   1:  PR[91,1] = PR[90,1] + 59.644;
   1:  PR[91,2] = PR[90,2] + 8.056;
   1:  PR[91,3] = PR[90,3] + 97.150;
   1:L PR[91] R[100]mm/sec CNT100;
   1:  PR[91,1] = PR[90,1] + 59.343;
   1:  PR[91,2] = PR[90,2] + 9.296;
   1:  PR[91,3] = PR[90,3] + 97.167;
   1:L PR[91] R[100]mm/sec CNT100;
   1:  PR[91,1] = PR[90,1] + 57.287;
   1:  PR[91,2] = PR[90,2] + 13.968;
   1:  PR[91,3] = PR[90,3] + 97.173;
   1:L PR[91] R[100]mm/sec CNT100;
   1:  PR[91,1] = PR[90,1] + 55.950;
   1:  PR[91,2] = PR[90,2] + 15.985;
   1:  PR[91,3] = PR[90,3] + 97.197;
   1:L PR[91] R[100]mm/sec CNT100;
   1:  PR[91,1] = PR[90,1] + 54.623;
   1:  PR[91,2] = PR[90,2] + 18.068;
   1:  PR[91,3] = PR[90,3] + 97.208;
   1:L PR[91] R[100]mm/sec CNT100;
   1:  PR[91,1] = PR[90,1] + 54.429;
   1:  PR[91,2] = PR[90,2] + 18.332;
   1:  PR[91,3] = PR[90,3] + 97.219;
   1:L PR[91] R[100]mm/sec CNT100;
   1:  PR[91,1] = PR[90,1] + 51.627;
   1:  PR[91,2] = PR[90,2] + 21.412;
   1:  PR[91,3] = PR[90,3] + 97.221;
   1:L PR[91] R[100]mm/sec CNT100;
   1:  PR[91,1] = PR[90,1] + 50.703;
   1:  PR[91,2] = PR[90,2] + 22.281;
   1:  PR[91,3] = PR[90,3] + 97.240;
   1:L PR[91] R[100]mm/sec CNT100;
   1:  PR[91,1] = PR[90,1] + 47.984;
   1:  PR[91,2] = PR[90,2] + 24.384;
   1:  PR[91,3] = PR[90,3] + 97.245;
   1:L PR[91] R[100]mm/sec CNT100;
   1:  PR[91,1] = PR[90,1] + 46.221;
   1:  PR[91,2] = PR[90,2] + 25.519;
   1:  PR[91,3] = PR[90,3] + 97.261;
   1:L PR[91] R[100]mm/sec CNT100;
   1:  PR[91,1] = PR[90,1] + 43.733;
   1:  PR[91,2] = PR[90,2] + 26.821;
   1:  PR[91,3] = PR[90,3] + 97.271;
   1:L PR[91] R[100]mm/sec CNT100;
   1:  PR[91,1] = PR[90,1] + 41.141;
   1:  PR[91,2] = PR[90,2] + 27.881;
   1:  PR[91,3] = PR[90,3] + 97.284;
   1:L PR[91] R[100]mm/sec CNT100;
   1:  PR[91,1] = PR[90,1] + 38.967;
   1:  PR[91,2] = PR[90,2] + 28.562;
   1:  PR[91,3] = PR[90,3] + 97.296;
   1:L PR[91] R[100]mm/sec CNT100;
   1:  PR[91,1] = PR[90,1] + 35.650;
   1:  PR[91,2] = PR[90,2] + 29.250;
   1:  PR[91,3] = PR[90,3] + 97.307;
   1:L PR[91] R[100]mm/sec CNT100;
   1:  PR[91,1] = PR[90,1] + 33.828;
   1:  PR[91,2] = PR[90,2] + 29.479;
   1:  PR[91,3] = PR[90,3] + 97.322;
   1:L PR[91] R[100]mm/sec CNT100;
   1:  PR[91,1] = PR[90,1] + 29.961;
   1:  PR[91,2] = PR[90,2] + 29.556;
   1:  PR[91,3] = PR[90,3] + 97.331;
   1:L PR[91] R[100]mm/sec CNT100;
   1:  PR[91,1] = PR[90,1] + 28.489;
   1:  PR[91,2] = PR[90,2] + 29.474;
   1:  PR[91,3] = PR[90,3] + 97.348;
   1:L PR[91] R[100]mm/sec CNT100;
   1:  PR[91,1] = PR[90,1] + 24.336;
   1:  PR[91,2] = PR[90,2] + 28.801;
   1:  PR[91,3] = PR[90,3] + 97.355;
   1:L PR[91] R[100]mm/sec CNT100;
   1:  PR[91,1] = PR[90,1] + 22.553;
   1:  PR[91,2] = PR[90,2] + 28.380;
   1:  PR[91,3] = PR[90,3] + 97.374;
   1:L PR[91] R[100]mm/sec CNT100;
   1:  PR[91,1] = PR[90,1] + 19.478;
   1:  PR[91,2] = PR[90,2] + 28.435;
   1:  PR[91,3] = PR[90,3] + 97.383;
   1:L PR[91] R[100]mm/sec CNT100;
   1:  PR[91,1] = PR[90,1] + 13.914;
   1:  PR[91,2] = PR[90,2] + 28.656;
   1:  PR[91,3] = PR[90,3] + 97.397;
   1:L PR[91] R[100]mm/sec CNT100;
   1:  PR[91,1] = PR[90,1] + 4.658;
   1:  PR[91,2] = PR[90,2] + 28.213;
   1:  PR[91,3] = PR[90,3] + 97.422;
   1:L PR[91] R[100]mm/sec CNT100;
   1:  PR[91,1] = PR[90,1] + -5.612;
   1:  PR[91,2] = PR[90,2] + 27.093;
   1:  PR[91,3] = PR[90,3] + 97.465;
   1:L PR[91] R[100]mm/sec CNT100;
   1:  PR[91,1] = PR[90,1] + -15.183;
   1:  PR[91,2] = PR[90,2] + 25.356;
   1:  PR[91,3] = PR[90,3] + 97.512;
   1:L PR[91] R[100]mm/sec CNT100;
   1:  PR[91,1] = PR[90,1] + -20.066;
   1:  PR[91,2] = PR[90,2] + 24.087;
   1:  PR[91,3] = PR[90,3] + 97.556;
   1:L PR[91] R[100]mm/sec CNT100;
   1:  PR[91,1] = PR[90,1] + -23.878;
   1:  PR[91,2] = PR[90,2] + 23.078;
   1:  PR[91,3] = PR[90,3] + 97.579;
   1:L PR[91] R[100]mm/sec CNT100;
   1:  PR[91,1] = PR[90,1] + -31.581;
   1:  PR[91,2] = PR[90,2] + 20.332;
   1:  PR[91,3] = PR[90,3] + 97.597;
   1:L PR[91] R[100]mm/sec CNT100;
   1:  PR[91,1] = PR[90,1] + -38.178;
   1:  PR[91,2] = PR[90,2] + 17.213;
   1:  PR[91,3] = PR[90,3] + 97.635;
   1:L PR[91] R[100]mm/sec CNT100;
   1:  PR[91,1] = PR[90,1] + -38.338;
   1:  PR[91,2] = PR[90,2] + 17.112;
   1:  PR[91,3] = PR[90,3] + 97.668;
   1:L PR[91] R[100]mm/sec CNT100;
   1:  PR[91,1] = PR[90,1] + -43.000;
   1:  PR[91,2] = PR[90,2] + 13.888;
   1:  PR[91,3] = PR[90,3] + 97.669;
   1:L PR[91] R[100]mm/sec CNT100;
   1:  PR[91] = PR[90];
   1:  PR[91,1] = PR[90,1] + -45.475;
   1:  PR[91,2] = PR[90,2] + 9.692;
   1:  PR[91,3] = PR[90,3] + 98.995;
   1:L PR[91] R[100]mm/sec CNT100;
   1:  PR[91,1] = PR[90,1] + -46.506;
   1:  PR[91,2] = PR[90,2] + 8.278;
   1:  PR[91,3] = PR[90,3] + 97.715;
   1:L PR[91] R[100]mm/sec CNT100;
   1:  PR[91,1] = PR[90,1] + -48.544;
   1:  PR[91,2] = PR[90,2] + 4.636;
   1:  PR[91,3] = PR[90,3] + 97.723;
   1:L PR[91] R[100]mm/sec CNT100;
   1:  PR[91,1] = PR[90,1] + -48.789;
   1:  PR[91,2] = PR[90,2] + 4.059;
   1:  PR[91,3] = PR[90,3] + 97.742;
   1:L PR[91] R[100]mm/sec CNT100;
   1:  PR[91,1] = PR[90,1] + -49.633;
   1:  PR[91,2] = PR[90,2] + -0.522;
   1:  PR[91,3] = PR[90,3] + 97.745;
   1:L PR[91] R[100]mm/sec CNT100;
   1:  PR[91,1] = PR[90,1] + -49.652;
   1:  PR[91,2] = PR[90,2] + -0.655;
   1:  PR[91,3] = PR[90,3] + 97.766;
   1:L PR[91] R[100]mm/sec CNT100;
   1:  PR[91,1] = PR[90,1] + -48.823;
   1:  PR[91,2] = PR[90,2] + -4.526;
   1:  PR[91,3] = PR[90,3] + 97.767;
   1:L PR[91] R[100]mm/sec CNT100;
   1:  PR[91,1] = PR[90,1] + -48.697;
   1:  PR[91,2] = PR[90,2] + -5.464;
   1:  PR[91,3] = PR[90,3] + 97.785;
   1:L PR[91] R[100]mm/sec CNT100;
   1:  PR[91,1] = PR[90,1] + -48.310;
   1:  PR[91,2] = PR[90,2] + -6.384;
   1:  PR[91,3] = PR[90,3] + 97.790;
   1:L PR[91] R[100]mm/sec CNT100;
   1:  PR[91,1] = PR[90,1] + -46.512;
   1:  PR[91,2] = PR[90,2] + -9.602;
   1:  PR[91,3] = PR[90,3] + 97.794;
   1:L PR[91] R[100]mm/sec CNT100;
   1:  PR[91,1] = PR[90,1] + -45.298;
   1:  PR[91,2] = PR[90,2] + -11.285;
   1:  PR[91,3] = PR[90,3] + 97.811;
   1:L PR[91] R[100]mm/sec CNT100;
   1:  PR[91,1] = PR[90,1] + -43.541;
   1:  PR[91,2] = PR[90,2] + -13.068;
   1:  PR[91,3] = PR[90,3] + 97.821;
   1:L PR[91] R[100]mm/sec CNT100;
   1:  PR[91,1] = PR[90,1] + -41.041;
   1:  PR[91,2] = PR[90,2] + -15.464;
   1:  PR[91,3] = PR[90,3] + 97.832;
   1:L PR[91] R[100]mm/sec CNT100;
   1:  PR[91,1] = PR[90,1] + -38.983;
   1:  PR[91,2] = PR[90,2] + -16.899;
   1:  PR[91,3] = PR[90,3] + 97.848;
   1:L PR[91] R[100]mm/sec CNT100;
   1:  PR[91,1] = PR[90,1] + -35.940;
   1:  PR[91,2] = PR[90,2] + -18.820;
   1:  PR[91,3] = PR[90,3] + 97.860;
   1:L PR[91] R[100]mm/sec CNT100;
   1:  PR[91,1] = PR[90,1] + -29.296;
   1:  PR[91,2] = PR[90,2] + -21.964;
   1:  PR[91,3] = PR[90,3] + 97.877;
   1:L PR[91] R[100]mm/sec CNT100;
   1:  PR[91,1] = PR[90,1] + -21.539;
   1:  PR[91,2] = PR[90,2] + -24.732;
   1:  PR[91,3] = PR[90,3] + 97.911;
   1:L PR[91] R[100]mm/sec CNT100;
   1:  PR[91,1] = PR[90,1] + -16.949;
   1:  PR[91,2] = PR[90,2] + -25.948;
   1:  PR[91,3] = PR[90,3] + 97.949;
   1:L PR[91] R[100]mm/sec CNT100;
   1:  PR[91,1] = PR[90,1] + -12.780;
   1:  PR[91,2] = PR[90,2] + -27.031;
   1:  PR[91,3] = PR[90,3] + 97.971;
   1:L PR[91] R[100]mm/sec CNT100;
   1:  PR[91,1] = PR[90,1] + -5.199;
   1:  PR[91,2] = PR[90,2] + -28.417;
   1:  PR[91,3] = PR[90,3] + 97.991;
   1:L PR[91] R[100]mm/sec CNT100;
   1:  PR[91,1] = PR[90,1] + -3.145;
   1:  PR[91,2] = PR[90,2] + -28.783;
   1:  PR[91,3] = PR[90,3] + 98.026;
   1:L PR[91] R[100]mm/sec CNT100;
   1:  PR[91,1] = PR[90,1] + 5.106;
   1:  PR[91,2] = PR[90,2] + -29.684;
   1:  PR[91,3] = PR[90,3] + 98.036;
   1:L PR[91] R[100]mm/sec CNT100;
